LIN {X 0,Y 445.914,Z 450.872,A -85,B 0,C 180,E1 -16893.892,E2 -16893.892} C_VEL
LIN {X 0,Y 439.308,Z 442.238,A -85,B 0,C 180,E1 -16896.064,E2 -16896.064} C_VEL
LIN {X 0,Y 435.286,Z 437.114,A -85,B 0,C 180,E1 -16897.513,E2 -16897.513} C_VEL
LIN {X 0,Y 431.118,Z 431.872,A -85,B 0,C 180,E1 -16899.144,E2 -16899.144} C_VEL
LIN {X 0,Y 426.688,Z 426.377,A -85,B 0,C 180,E1 -16901.061,E2 -16901.061} C_VEL
LIN {X 0,Y 423.049,Z 422.011,A -85,B 0,C 180,E1 -16902.816,E2 -16902.816} C_VEL
LIN {X 0,Y 422.048,Z 420.717,A -85,B 0,C 180,E1 -16903.341,E2 -16903.341} C_VEL
LIN {X 0,Y 418.805,Z 417.442,A -85,B 0,C 180,E1 -16905.128,E2 -16905.128} C_VEL
LIN {X 0,Y 417.28,Z 414.785,A -85,B 0,C 180,E1 -16906.136,E2 -16906.136} C_VEL
LIN {X 0,Y 413.911,Z 412.07,A -85,B 0,C 180,E1 -16908.434,E2 -16908.434} C_VEL
LIN {X 0,Y 411.982,Z 408.411,A -85,B 0,C 180,E1 -16910.218,E2 -16910.218} C_VEL
LIN {X 0,Y 408.184,Z 405.747,A -85,B 0,C 180,E1 -16914.659,E2 -16914.659} C_VEL
LIN {X 0,Y 406.884,Z 403.015,A -85,B 0,C 180,E1 -16919.155,E2 -16919.155} C_VEL
LIN {X 0,Y 406.916,Z 403.188,A -85,B 0,C 180,E1 -16920.986,E2 -16920.986} C_VEL
LIN {X 0,Y 411.873,Z 408.41,A -85,B 0,C 180,E1 -16929.361,E2 -16929.361} C_VEL
LIN {X 0,Y 414.509,Z 412.704,A -85,B 0,C 180,E1 -16931.691,E2 -16931.691} C_VEL
LIN {X 0,Y 417.544,Z 415.253,A -85,B 0,C 180,E1 -16933.714,E2 -16933.714} C_VEL
LIN {X 0,Y 420.375,Z 419.282,A -85,B 0,C 180,E1 -16935.45,E2 -16935.45} C_VEL
LIN {X 0,Y 422.697,Z 421.438,A -85,B 0,C 180,E1 -16936.664,E2 -16936.664} C_VEL
LIN {X 0,Y 425.915,Z 425.709,A -85,B 0,C 180,E1 -16938.265,E2 -16938.265} C_VEL
LIN {X 0,Y 427.713,Z 427.589,A -85,B 0,C 180,E1 -16939.069,E2 -16939.069} C_VEL
LIN {X 0,Y 431.546,Z 432.247,A -85,B 0,C 180,E1 -16940.692,E2 -16940.692} C_VEL
LIN {X 0,Y 438.177,Z 440.986,A -85,B 0,C 180,E1 -16943.216,E2 -16943.216} C_VEL
LIN {X 0,Y 447.328,Z 454.311,A -85,B 0,C 180,E1 -16946.269,E2 -16946.269} C_VEL
LIN {X 0,Y 457.218,Z 469.808,A -85,B 0,C 180,E1 -16949.152,E2 -16949.152} C_VEL
LIN {X 0,Y 466.824,Z 485.963,A -85,B 0,C 180,E1 -16951.653,E2 -16951.653} C_VEL
LIN {X 0,Y 475.146,Z 500.955,A -85,B 0,C 180,E1 -16953.636,E2 -16953.636} C_VEL
LIN {X 0,Y 460.946,Z 747.179,A -85,B 0,C 180,E1 -16957.557,E2 -16957.557} C_VEL
LIN {X 0,Y 458.843,Z 772.183,A -85,B 0,C 180,E1 -16958.029,E2 -16958.029} C_VEL
LIN {X 0,Y 455.888,Z 795.416,A -85,B 0,C 180,E1 -16958.602,E2 -16958.602} C_VEL
LIN {X 0,Y 451.88,Z 819.021,A -85,B 0,C 180,E1 -16959.383,E2 -16959.383} C_VEL
LIN {X 0,Y 448.092,Z 837.848,A -85,B 0,C 180,E1 -16960.157,E2 -16960.157} C_VEL
LIN {X 0,Y 442.735,Z 861.158,A -85,B 0,C 180,E1 -16961.329,E2 -16961.329} C_VEL
LIN {X 0,Y 437.251,Z 881.76,A -85,B 0,C 180,E1 -16962.601,E2 -16962.601} C_VEL
LIN {X 0,Y 431.383,Z 901.908,A -85,B 0,C 180,E1 -16964.066,E2 -16964.066} C_VEL
LIN {X 0,Y 424.657,Z 922.896,A -85,B 0,C 180,E1 -16965.902,E2 -16965.902} C_VEL
LIN {X 0,Y 418.742,Z 940.201,A -85,B 0,C 180,E1 -16967.672,E2 -16967.672} C_VEL
LIN {X 0,Y 411.479,Z 960.285,A -85,B 0,C 180,E1 -16970.095,E2 -16970.095} C_VEL
LIN {X 0,Y 405.621,Z 975.927,A -85,B 0,C 180,E1 -16972.313,E2 -16972.313} C_VEL
LIN {X 0,Y 398.802,Z 993.871,A -85,B 0,C 180,E1 -16975.309,E2 -16975.309} C_VEL
LIN {X 0,Y 393.732,Z 1007.261,A -85,B 0,C 180,E1 -16977.943,E2 -16977.943} C_VEL
LIN {X 0,Y 388.289,Z 1022.091,A -85,B 0,C 180,E1 -16981.382,E2 -16981.382} C_VEL
LIN {X 0,Y 384.646,Z 1032.615,A -85,B 0,C 180,E1 -16984.271,E2 -16984.271} C_VEL
LIN {X 0,Y 381.229,Z 1043.573,A -85,B 0,C 180,E1 -16987.81,E2 -16987.81} C_VEL
LIN {X 0,Y 378.881,Z 1052.198,A -85,B 0,C 180,E1 -16991.218,E2 -16991.218} C_VEL
LIN {X 0,Y 377.283,Z 1059.672,A -85,B 0,C 180,E1 -16994.789,E2 -16994.789} C_VEL
LIN {X 0,Y 376.39,Z 1065.338,A -85,B 0,C 180,E1 -16998.352,E2 -16998.352} C_VEL
LIN {X 0,Y 376.05,Z 1069.072,A -85,B 0,C 180,E1 -17001.437,E2 -17001.437} C_VEL
LIN {X 0,Y 375.953,Z 1072.023,A -85,B 0,C 180,E1 -17004.965,E2 -17004.965} C_VEL
LIN {X 0,Y 375.957,Z 1073.297,A -85,B 0,C 180,E1 -17008.323,E2 -17008.323} C_VEL
LIN {X 0,Y 375.964,Z 1073.365,A -85,B 0,C 180,E1 -17011.219,E2 -17011.219} C_VEL
LIN {X 0,Y 375.948,Z 1072.423,A -85,B 0,C 180,E1 -17014.152,E2 -17014.152} C_VEL
LIN {X 0,Y 375.991,Z 1070.035,A -85,B 0,C 180,E1 -17017.641,E2 -17017.641} C_VEL
LIN {X 0,Y 376.318,Z 1065.955,A -85,B 0,C 180,E1 -17021.184,E2 -17021.184} C_VEL
LIN {X 0,Y 377.033,Z 1060.963,A -85,B 0,C 180,E1 -17024.435,E2 -17024.435} C_VEL
LIN {X 0,Y 378.625,Z 1053.245,A -85,B 0,C 180,E1 -17028.316,E2 -17028.316} C_VEL
LIN {X 0,Y 380.724,Z 1045.185,A -85,B 0,C 180,E1 -17031.572,E2 -17031.572} C_VEL
LIN {X 0,Y 383.966,Z 1034.661,A -85,B 0,C 180,E1 -17035.117,E2 -17035.117} C_VEL
LIN {X 0,Y 387.657,Z 1023.784,A -85,B 0,C 180,E1 -17038.165,E2 -17038.165} C_VEL
LIN {X 0,Y 392.448,Z 1010.715,A -85,B 0,C 180,E1 -17041.316,E2 -17041.316} C_VEL
LIN {X 0,Y 397.898,Z 996.124,A -85,B 0,C 180,E1 -17044.256,E2 -17044.256} C_VEL
LIN {X 0,Y 403.578,Z 981.252,A -85,B 0,C 180,E1 -17046.845,E2 -17046.845} C_VEL
LIN {X 0,Y 410.123,Z 963.744,A -85,B 0,C 180,E1 -17049.428,E2 -17049.428} C_VEL
LIN {X 0,Y 416.214,Z 947.095,A -85,B 0,C 180,E1 -17051.532,E2 -17051.532} C_VEL
LIN {X 0,Y 423.277,Z 926.792,A -85,B 0,C 180,E1 -17053.709,E2 -17053.709} C_VEL
LIN {X 0,Y 429.253,Z 908.409,A -85,B 0,C 180,E1 -17055.382,E2 -17055.382} C_VEL
LIN {X 0,Y 436.027,Z 885.844,A -85,B 0,C 180,E1 -17057.111,E2 -17057.111} C_VEL
LIN {X 0,Y 441.133,Z 866.944,A -85,B 0,C 180,E1 -17058.319,E2 -17058.319} C_VEL
LIN {X 0,Y 446.428,Z 845.202,A -85,B 0,C 180,E1 -17059.494,E2 -17059.494} C_VEL
LIN {X 0,Y 451.109,Z 822.479,A -85,B 0,C 180,E1 -17060.475,E2 -17060.475} C_VEL
LIN {X 0,Y 454.909,Z 800.788,A -85,B 0,C 180,E1 -17061.227,E2 -17061.227} C_VEL
LIN {X 0,Y 458.427,Z 774.973,A -85,B 0,C 180,E1 -17061.899,E2 -17061.899} C_VEL
LIN {X 0,Y 460.452,Z 752.549,A -85,B 0,C 180,E1 -17062.338,E2 -17062.338} C_VEL
LIN {X 0,Y 474.798,Z 504.728,A -85,B 0,C 180,E1 -17066.292,E2 -17066.292} C_VEL
LIN {X 0,Y 474.918,Z 500.686,A -85,B 0,C 180,E1 -17066.377,E2 -17066.377} C_VEL
LIN {X 0,Y 465.136,Z 483.112,A -85,B 0,C 180,E1 -17068.725,E2 -17068.725} C_VEL
LIN {X 0,Y 455.822,Z 467.629,A -85,B 0,C 180,E1 -17071.181,E2 -17071.181} C_VEL
LIN {X 0,Y 446.583,Z 453.314,A -85,B 0,C 180,E1 -17073.899,E2 -17073.899} C_VEL
LIN {X 0,Y 439.183,Z 442.658,A -85,B 0,C 180,E1 -17076.342,E2 -17076.342} C_VEL
LIN {X 0,Y 435.375,Z 437.187,A -85,B 0,C 180,E1 -17077.732,E2 -17077.732} C_VEL
LIN {X 0,Y 431.177,Z 431.925,A -85,B 0,C 180,E1 -17079.361,E2 -17079.361} C_VEL
LIN {X 0,Y 427.435,Z 427.213,A -85,B 0,C 180,E1 -17080.954,E2 -17080.954} C_VEL
LIN {X 0,Y 423.28,Z 422.498,A -85,B 0,C 180,E1 -17082.896,E2 -17082.896} C_VEL
LIN {X 0,Y 422.163,Z 420.799,A -85,B 0,C 180,E1 -17083.488,E2 -17083.488} C_VEL
LIN {X 0,Y 418.647,Z 417.219,A -85,B 0,C 180,E1 -17085.406,E2 -17085.406} C_VEL
LIN {X 0,Y 417.091,Z 414.724,A -85,B 0,C 180,E1 -17086.412,E2 -17086.412} C_VEL
LIN {X 0,Y 413.807,Z 411.904,A -85,B 0,C 180,E1 -17088.642,E2 -17088.642} C_VEL
LIN {X 0,Y 411.904,Z 408.425,A -85,B 0,C 180,E1 -17090.358,E2 -17090.358} C_VEL
LIN {X 0,Y 407.764,Z 405.265,A -85,B 0,C 180,E1 -17095.218,E2 -17095.218} C_VEL
LIN {X 0,Y 406.659,Z 401.868,A -85,B 0,C 180,E1 -17099.577,E2 -17099.577} C_VEL
LIN {X 0,Y 406.701,Z 402.227,A -85,B 0,C 180,E1 -17101.55,E2 -17101.55} C_VEL
LIN {X 0,Y 410.534,Z 407.839,A -85,B 0,C 180,E1 -17108.826,E2 -17108.826} C_VEL
LIN {X 0,Y 412.126,Z 408.762,A -85,B 0,C 180,E1 -17110.272,E2 -17110.272} C_VEL
LIN {X 0,Y 414.158,Z 412.402,A -85,B 0,C 180,E1 -17112.054,E2 -17112.054} C_VEL
LIN {X 0,Y 417.516,Z 415.258,A -85,B 0,C 180,E1 -17114.281,E2 -17114.281} C_VEL
LIN {X 0,Y 420.259,Z 419.245,A -85,B 0,C 180,E1 -17115.95,E2 -17115.95} C_VEL
LIN {X 0,Y 422.739,Z 421.532,A -85,B 0,C 180,E1 -17117.233,E2 -17117.233} C_VEL
LIN {X 0,Y 426.281,Z 426.044,A -85,B 0,C 180,E1 -17118.958,E2 -17118.958} C_VEL
LIN {X 0,Y 427.727,Z 427.665,A -85,B 0,C 180,E1 -17119.6,E2 -17119.6} C_VEL
LIN {X 0,Y 431.51,Z 432.267,A -85,B 0,C 180,E1 -17121.191,E2 -17121.191} C_VEL
LIN {X 0,Y 437.246,Z 439.664,A -85,B 0,C 180,E1 -17123.376,E2 -17123.376} C_VEL
LIN {X 0,Y 441.857,Z 445.634,A -85,B 0,C 180,E1 -17124.963,E2 -17124.963} C_VEL
LIN {X 0,Y 448.316,Z 454.069,A -85,B 0,C 180,E1 -17126.992,E2 -17126.992} C_VEL
LIN {X 0,Y 458.368,Z 468.203,A -85,B 0,C 180,E1 -17129.826,E2 -17129.826} C_VEL
LIN {X 0,Y 467.534,Z 481.985,A -85,B 0,C 180,E1 -17132.14,E2 -17132.14} C_VEL
LIN {X 0,Y 475.238,Z 494.264,A -85,B 0,C 180,E1 -17133.93,E2 -17133.93} C_VEL
LIN {X 0,Y 460.96,Z 738.871,A -85,B 0,C 180,E1 -17137.83,E2 -17137.83} C_VEL
LIN {X 0,Y 458.981,Z 760.833,A -85,B 0,C 180,E1 -17138.272,E2 -17138.272} C_VEL
LIN {X 0,Y 455.614,Z 786.437,A -85,B 0,C 180,E1 -17138.98,E2 -17138.98} C_VEL
LIN {X 0,Y 452.234,Z 806.44,A -85,B 0,C 180,E1 -17139.698,E2 -17139.698} C_VEL
LIN {X 0,Y 447.751,Z 829.084,A -85,B 0,C 180,E1 -17140.699,E2 -17140.699} C_VEL
LIN {X 0,Y 442.594,Z 850.765,A -85,B 0,C 180,E1 -17141.893,E2 -17141.893} C_VEL
LIN {X 0,Y 437.114,Z 871.313,A -85,B 0,C 180,E1 -17143.234,E2 -17143.234} C_VEL
LIN {X 0,Y 430.715,Z 892.744,A -85,B 0,C 180,E1 -17144.924,E2 -17144.924} C_VEL
LIN {X 0,Y 424.856,Z 910.758,A -85,B 0,C 180,E1 -17146.59,E2 -17146.59} C_VEL
LIN {X 0,Y 417.698,Z 931.227,A -85,B 0,C 180,E1 -17148.83,E2 -17148.83} C_VEL
LIN {X 0,Y 411.851,Z 947.019,A -85,B 0,C 180,E1 -17150.86,E2 -17150.86} C_VEL
LIN {X 0,Y 405.104,Z 964.603,A -85,B 0,C 180,E1 -17153.499,E2 -17153.499} C_VEL
LIN {X 0,Y 399.413,Z 979.074,A -85,B 0,C 180,E1 -17156.065,E2 -17156.065} C_VEL
LIN {X 0,Y 393.645,Z 993.854,A -85,B 0,C 180,E1 -17159.13,E2 -17159.13} C_VEL
LIN {X 0,Y 388.99,Z 1005.906,A -85,B 0,C 180,E1 -17162.107,E2 -17162.107} C_VEL
LIN {X 0,Y 384.833,Z 1017.408,A -85,B 0,C 180,E1 -17165.436,E2 -17165.436} C_VEL
LIN {X 0,Y 381.521,Z 1027.213,A -85,B 0,C 180,E1 -17168.909,E2 -17168.909} C_VEL
LIN {X 0,Y 379.086,Z 1035.65,A -85,B 0,C 180,E1 -17172.501,E2 -17172.501} C_VEL
LIN {X 0,Y 377.492,Z 1042.13,A -85,B 0,C 180,E1 -17176.052,E2 -17176.052} C_VEL
LIN {X 0,Y 376.627,Z 1046.785,A -85,B 0,C 180,E1 -17179.29,E2 -17179.29} C_VEL
LIN {X 0,Y 376.148,Z 1050.669,A -85,B 0,C 180,E1 -17183.13,E2 -17183.13} C_VEL
LIN {X 0,Y 376.009,Z 1052.533,A -85,B 0,C 180,E1 -17186.188,E2 -17186.188} C_VEL
LIN {X 0,Y 375.969,Z 1053.36,A -85,B 0,C 180,E1 -17189.238,E2 -17189.238} C_VEL
LIN {X 0,Y 375.985,Z 1053.045,A -85,B 0,C 180,E1 -17192.744,E2 -17192.744} C_VEL
LIN {X 0,Y 376.092,Z 1051.299,A -85,B 0,C 180,E1 -17196.105,E2 -17196.105} C_VEL
LIN {X 0,Y 376.366,Z 1048.637,A -85,B 0,C 180,E1 -17199.172,E2 -17199.172} C_VEL
LIN {X 0,Y 377.086,Z 1044.286,A -85,B 0,C 180,E1 -17202.714,E2 -17202.714} C_VEL
LIN {X 0,Y 378.398,Z 1038.227,A -85,B 0,C 180,E1 -17206.266,E2 -17206.266} C_VEL
LIN {X 0,Y 380.273,Z 1031.39,A -85,B 0,C 180,E1 -17209.508,E2 -17209.508} C_VEL
LIN {X 0,Y 383.325,Z 1021.762,A -85,B 0,C 180,E1 -17213.196,E2 -17213.196} C_VEL
LIN {X 0,Y 386.688,Z 1012.189,A -85,B 0,C 180,E1 -17216.242,E2 -17216.242} C_VEL
LIN {X 0,Y 388.467,Z 1007.407,A -85,B 0,C 180,E1 -17217.598,E2 -17217.598} C_VEL
LIN {X 0,Y 388.905,Z 1003.88,A -85,B 0,C 180,E1 -17218.615,E2 -17218.615} C_VEL
LIN {X 0,Y 387.122,Z 994.607,A -85,B 0,C 180,E1 -17221.427,E2 -17221.427} C_VEL
LIN {X 0,Y 387.838,Z 991.149,A -85,B 0,C 180,E1 -17222.262,E2 -17222.262} C_VEL
LIN {X 0,Y 393.105,Z 978.251,A -85,B 0,C 180,E1 -17224.911,E2 -17224.911} C_VEL
LIN {X 0,Y 399.46,Z 962.832,A -85,B 0,C 180,E1 -17227.644,E2 -17227.644} C_VEL
LIN {X 0,Y 406.146,Z 945.85,A -85,B 0,C 180,E1 -17230.167,E2 -17230.167} C_VEL
LIN {X 0,Y 412.721,Z 928.691,A -85,B 0,C 180,E1 -17232.36,E2 -17232.36} C_VEL
LIN {X 0,Y 419.697,Z 909.139,A -85,B 0,C 180,E1 -17234.462,E2 -17234.462} C_VEL
LIN {X 0,Y 425.918,Z 890.53,A -85,B 0,C 180,E1 -17236.168,E2 -17236.168} C_VEL
LIN {X 0,Y 432.407,Z 869.027,A -85,B 0,C 180,E1 -17237.827,E2 -17237.827} C_VEL
LIN {X 0,Y 437.827,Z 849.172,A -85,B 0,C 180,E1 -17239.106,E2 -17239.106} C_VEL
LIN {X 0,Y 443.66,Z 824.456,A -85,B 0,C 180,E1 -17240.424,E2 -17240.424} C_VEL
LIN {X 0,Y 447.87,Z 803.378,A -85,B 0,C 180,E1 -17241.327,E2 -17241.327} C_VEL
LIN {X 0,Y 452.017,Z 777.908,A -85,B 0,C 180,E1 -17242.186,E2 -17242.186} C_VEL
LIN {X 0,Y 454.733,Z 755.827,A -85,B 0,C 180,E1 -17242.742,E2 -17242.742} C_VEL
LIN {X 0,Y 456.958,Z 728.166,A -85,B 0,C 180,E1 -17243.252,E2 -17243.252} C_VEL
LIN {X 0,Y 470.68,Z 498.278,A -85,B 0,C 180,E1 -17246.928,E2 -17246.928} C_VEL
LIN {X 0,Y 460.809,Z 482.688,A -85,B 0,C 180,E1 -17249.342,E2 -17249.342} C_VEL
LIN {X 0,Y 451.523,Z 469.038,A -85,B 0,C 180,E1 -17251.856,E2 -17251.856} C_VEL
LIN {X 0,Y 443.324,Z 457.626,A -85,B 0,C 180,E1 -17254.339,E2 -17254.339} C_VEL
LIN {X 0,Y 436.928,Z 449.186,A -85,B 0,C 180,E1 -17256.499,E2 -17256.499} C_VEL
LIN {X 0,Y 433.152,Z 444.297,A -85,B 0,C 180,E1 -17257.897,E2 -17257.897} C_VEL
LIN {X 0,Y 429.218,Z 439.263,A -85,B 0,C 180,E1 -17259.476,E2 -17259.476} C_VEL
LIN {X 0,Y 425.01,Z 433.941,A -85,B 0,C 180,E1 -17261.34,E2 -17261.34} C_VEL
LIN {X 0,Y 421.316,Z 429.373,A -85,B 0,C 180,E1 -17263.17,E2 -17263.17} C_VEL
LIN {X 0,Y 420.319,Z 428.242,A -85,B 0,C 180,E1 -17263.697,E2 -17263.697} C_VEL
LIN {X 0,Y 417.071,Z 424.661,A -85,B 0,C 180,E1 -17265.562,E2 -17265.562} C_VEL
LIN {X 0,Y 415.885,Z 422.55,A -85,B 0,C 180,E1 -17266.372,E2 -17266.372} C_VEL
LIN {X 0,Y 412.595,Z 419.762,A -85,B 0,C 180,E1 -17268.679,E2 -17268.679} C_VEL
LIN {X 0,Y 410.702,Z 416.259,A -85,B 0,C 180,E1 -17270.471,E2 -17270.471} C_VEL
LIN {X 0,Y 406.544,Z 412.767,A -85,B 0,C 180,E1 -17276.051,E2 -17276.051} C_VEL
LIN {X 0,Y 405.909,Z 410.957,A -85,B 0,C 180,E1 -17279.153,E2 -17279.153} C_VEL
LIN {X 0,Y 405.928,Z 411.083,A -85,B 0,C 180,E1 -17280.847,E2 -17280.847} C_VEL
LIN {X 0,Y 410.888,Z 416.54,A -85,B 0,C 180,E1 -17289.384,E2 -17289.384} C_VEL
LIN {X 0,Y 413,Z 420.204,A -85,B 0,C 180,E1 -17291.309,E2 -17291.309} C_VEL
LIN {X 0,Y 416.144,Z 423,A -85,B 0,C 180,E1 -17293.478,E2 -17293.478} C_VEL
LIN {X 0,Y 419.168,Z 427.21,A -85,B 0,C 180,E1 -17295.354,E2 -17295.354} C_VEL
LIN {X 0,Y 421.152,Z 429.131,A -85,B 0,C 180,E1 -17296.411,E2 -17296.411} C_VEL
LIN {X 0,Y 424.53,Z 433.532,A -85,B 0,C 180,E1 -17298.113,E2 -17298.113} C_VEL
LIN {X 0,Y 426.083,Z 435.288,A -85,B 0,C 180,E1 -17298.825,E2 -17298.825} C_VEL
LIN {X 0,Y 430.863,Z 441.312,A -85,B 0,C 180,E1 -17300.869,E2 -17300.869} C_VEL
LIN {X 0,Y 436.072,Z 448.276,A -85,B 0,C 180,E1 -17302.871,E2 -17302.871} C_VEL
LIN {X 0,Y 444.894,Z 461.347,A -85,B 0,C 180,E1 -17305.886,E2 -17305.886} C_VEL
LIN {X 0,Y 454.529,Z 476.71,A -85,B 0,C 180,E1 -17308.765,E2 -17308.765} C_VEL
LIN {X 0,Y 463.774,Z 492.562,A -85,B 0,C 180,E1 -17311.233,E2 -17311.233} C_VEL
LIN {X 0,Y 470.494,Z 504.94,A -85,B 0,C 180,E1 -17312.89,E2 -17312.89} C_VEL
LIN {X 0,Y 455.687,Z 752.602,A -85,B 0,C 180,E1 -17316.856,E2 -17316.856} C_VEL
LIN {X 0,Y 453.608,Z 774.959,A -85,B 0,C 180,E1 -17317.295,E2 -17317.295} C_VEL
LIN {X 0,Y 449.936,Z 801.11,A -85,B 0,C 180,E1 -17317.979,E2 -17317.979} C_VEL
LIN {X 0,Y 446.231,Z 821.754,A -85,B 0,C 180,E1 -17318.695,E2 -17318.695} C_VEL
LIN {X 0,Y 441.541,Z 844.082,A -85,B 0,C 180,E1 -17319.651,E2 -17319.651} C_VEL
LIN {X 0,Y 436.07,Z 865.993,A -85,B 0,C 180,E1 -17320.828,E2 -17320.828} C_VEL
LIN {X 0,Y 430.554,Z 885.873,A -85,B 0,C 180,E1 -17322.099,E2 -17322.099} C_VEL
LIN {X 0,Y 423.78,Z 907.768,A -85,B 0,C 180,E1 -17323.781,E2 -17323.781} C_VEL
LIN {X 0,Y 417.835,Z 925.512,A -85,B 0,C 180,E1 -17325.396,E2 -17325.396} C_VEL
LIN {X 0,Y 410.636,Z 945.656,A -85,B 0,C 180,E1 -17327.545,E2 -17327.545} C_VEL
LIN {X 0,Y 404.194,Z 962.624,A -85,B 0,C 180,E1 -17329.692,E2 -17329.692} C_VEL
LIN {X 0,Y 397.689,Z 979.441,A -85,B 0,C 180,E1 -17332.159,E2 -17332.159} C_VEL
LIN {X 0,Y 391.391,Z 995.21,A -85,B 0,C 180,E1 -17334.914,E2 -17334.914} C_VEL
LIN {X 0,Y 385.92,Z 1009.168,A -85,B 0,C 180,E1 -17337.742,E2 -17337.742} C_VEL
LIN {X 0,Y 380.726,Z 1022.659,A -85,B 0,C 180,E1 -17340.992,E2 -17340.992} C_VEL
LIN {X 0,Y 376.742,Z 1033.729,A -85,B 0,C 180,E1 -17344.122,E2 -17344.122} C_VEL
LIN {X 0,Y 373.191,Z 1044.59,A -85,B 0,C 180,E1 -17347.804,E2 -17347.804} C_VEL
LIN {X 0,Y 370.916,Z 1052.699,A -85,B 0,C 180,E1 -17351.126,E2 -17351.126} C_VEL
LIN {X 0,Y 369.175,Z 1060.507,A -85,B 0,C 180,E1 -17355.09,E2 -17355.09} C_VEL
LIN {X 0,Y 368.378,Z 1065.544,A -85,B 0,C 180,E1 -17358.413,E2 -17358.413} C_VEL
LIN {X 0,Y 368.014,Z 1069.51,A -85,B 0,C 180,E1 -17361.878,E2 -17361.878} C_VEL
LIN {X 0,Y 367.95,Z 1072.091,A -85,B 0,C 180,E1 -17365.48,E2 -17365.48} C_VEL
LIN {X 0,Y 367.963,Z 1073.13,A -85,B 0,C 180,E1 -17368.598,E2 -17368.598} C_VEL
LIN {X 0,Y 367.963,Z 1073.128,A -85,B 0,C 180,E1 -17371.401,E2 -17371.401} C_VEL
LIN {X 0,Y 367.951,Z 1072.084,A -85,B 0,C 180,E1 -17374.52,E2 -17374.52} C_VEL
LIN {X 0,Y 368.026,Z 1069.332,A -85,B 0,C 180,E1 -17378.279,E2 -17378.279} C_VEL
LIN {X 0,Y 368.378,Z 1065.527,A -85,B 0,C 180,E1 -17381.587,E2 -17381.587} C_VEL
LIN {X 0,Y 369.173,Z 1060.484,A -85,B 0,C 180,E1 -17384.91,E2 -17384.91} C_VEL
LIN {X 0,Y 370.917,Z 1052.653,A -85,B 0,C 180,E1 -17388.879,E2 -17388.879} C_VEL
LIN {X 0,Y 373.188,Z 1044.552,A -85,B 0,C 180,E1 -17392.196,E2 -17392.196} C_VEL
LIN {X 0,Y 376.835,Z 1033.394,A -85,B 0,C 180,E1 -17395.964,E2 -17395.964} C_VEL
LIN {X 0,Y 380.796,Z 1022.397,A -85,B 0,C 180,E1 -17399.063,E2 -17399.063} C_VEL
LIN {X 0,Y 386.228,Z 1008.248,A -85,B 0,C 180,E1 -17402.438,E2 -17402.438} C_VEL
LIN {X 0,Y 391.38,Z 995.121,A -85,B 0,C 180,E1 -17405.087,E2 -17405.087} C_VEL
LIN {X 0,Y 397.755,Z 979.124,A -85,B 0,C 180,E1 -17407.875,E2 -17407.875} C_VEL
LIN {X 0,Y 404.373,Z 961.987,A -85,B 0,C 180,E1 -17410.379,E2 -17410.379} C_VEL
LIN {X 0,Y 411.394,Z 943.499,A -85,B 0,C 180,E1 -17412.696,E2 -17412.696} C_VEL
LIN {X 0,Y 418.071,Z 924.575,A -85,B 0,C 180,E1 -17414.68,E2 -17414.68} C_VEL
LIN {X 0,Y 424.248,Z 906.082,A -85,B 0,C 180,E1 -17416.349,E2 -17416.349} C_VEL
LIN {X 0,Y 431.041,Z 883.812,A -85,B 0,C 180,E1 -17418.027,E2 -17418.027} C_VEL
LIN {X 0,Y 436.285,Z 864.804,A -85,B 0,C 180,E1 -17419.23,E2 -17419.23} C_VEL
LIN {X 0,Y 442.064,Z 841.142,A -85,B 0,C 180,E1 -17420.47,E2 -17420.47} C_VEL
LIN {X 0,Y 446.283,Z 820.92,A -85,B 0,C 180,E1 -17421.324,E2 -17421.324} C_VEL
LIN {X 0,Y 450.329,Z 798.213,A -85,B 0,C 180,E1 -17422.098,E2 -17422.098} C_VEL
LIN {X 0,Y 453.635,Z 773.646,A -85,B 0,C 180,E1 -17422.722,E2 -17422.722} C_VEL
LIN {X 0,Y 455.717,Z 750.597,A -85,B 0,C 180,E1 -17423.168,E2 -17423.168} C_VEL
LIN {X 0,Y 470.369,Z 504.718,A -85,B 0,C 180,E1 -17427.103,E2 -17427.103} C_VEL
LIN {X 0,Y 461.156,Z 488.101,A -85,B 0,C 180,E1 -17429.393,E2 -17429.393} C_VEL
LIN {X 0,Y 452.739,Z 473.897,A -85,B 0,C 180,E1 -17431.687,E2 -17431.687} C_VEL
LIN {X 0,Y 443.971,Z 460.049,A -85,B 0,C 180,E1 -17434.343,E2 -17434.343} C_VEL
LIN {X 0,Y 435.136,Z 446.928,A -85,B 0,C 180,E1 -17437.398,E2 -17437.398} C_VEL
LIN {X 0,Y 429.267,Z 439.317,A -85,B 0,C 180,E1 -17439.692,E2 -17439.692} C_VEL
LIN {X 0,Y 424.878,Z 433.867,A -85,B 0,C 180,E1 -17441.618,E2 -17441.618} C_VEL
LIN {X 0,Y 421.348,Z 429.558,A -85,B 0,C 180,E1 -17443.348,E2 -17443.348} C_VEL
LIN {X 0,Y 420.422,Z 428.32,A -85,B 0,C 180,E1 -17443.843,E2 -17443.843} C_VEL
LIN {X 0,Y 416.907,Z 424.438,A -85,B 0,C 180,E1 -17445.84,E2 -17445.84} C_VEL
LIN {X 0,Y 415.691,Z 422.489,A -85,B 0,C 180,E1 -17446.649,E2 -17446.649} C_VEL
LIN {X 0,Y 412.399,Z 419.482,A -85,B 0,C 180,E1 -17448.957,E2 -17448.957} C_VEL
LIN {X 0,Y 410.616,Z 416.27,A -85,B 0,C 180,E1 -17450.61,E2 -17450.61} C_VEL
LIN {X 0,Y 406.578,Z 412.906,A -85,B 0,C 180,E1 -17455.628,E2 -17455.628} C_VEL
LIN {X 0,Y 405.68,Z 409.842,A -85,B 0,C 180,E1 -17459.576,E2 -17459.576} C_VEL
LIN {X 0,Y 405.712,Z 410.106,A -85,B 0,C 180,E1 -17461.412,E2 -17461.412} C_VEL
LIN {X 0,Y 409.428,Z 415.727,A -85,B 0,C 180,E1 -17468.709,E2 -17468.709} C_VEL
LIN {X 0,Y 410.848,Z 416.485,A -85,B 0,C 180,E1 -17470.021,E2 -17470.021} C_VEL
LIN {X 0,Y 412.915,Z 420.204,A -85,B 0,C 180,E1 -17471.878,E2 -17471.878} C_VEL
LIN {X 0,Y 416.11,Z 423.018,A -85,B 0,C 180,E1 -17474.046,E2 -17474.046} C_VEL
LIN {X 0,Y 418.931,Z 427.055,A -85,B 0,C 180,E1 -17475.789,E2 -17475.789} C_VEL
LIN {X 0,Y 421.124,Z 429.106,A -85,B 0,C 180,E1 -17476.945,E2 -17476.945} C_VEL
LIN {X 0,Y 424.749,Z 433.733,A -85,B 0,C 180,E1 -17478.744,E2 -17478.744} C_VEL
LIN {X 0,Y 426.232,Z 435.587,A -85,B 0,C 180,E1 -17479.422,E2 -17479.422} C_VEL
LIN {X 0,Y 430.751,Z 441.257,A -85,B 0,C 180,E1 -17481.338,E2 -17481.338} C_VEL
LIN {X 0,Y 435.325,Z 447.163,A -85,B 0,C 180,E1 -17483.091,E2 -17483.091} C_VEL
LIN {X 0,Y 439.784,Z 453.022,A -85,B 0,C 180,E1 -17484.658,E2 -17484.658} C_VEL
LIN {X 0,Y 446.154,Z 461.528,A -85,B 0,C 180,E1 -17486.702,E2 -17486.702} C_VEL
LIN {X 0,Y 455.667,Z 475.098,A -85,B 0,C 180,E1 -17489.442,E2 -17489.442} C_VEL
LIN {X 0,Y 464.596,Z 488.732,A -85,B 0,C 180,E1 -17491.75,E2 -17491.75} C_VEL
LIN {X 0,Y 470.567,Z 498.521,A -85,B 0,C 180,E1 -17493.185,E2 -17493.185} C_VEL
LIN {X 0,Y 456.03,Z 739.962,A -85,B 0,C 180,E1 -17497.051,E2 -17497.051} C_VEL
LIN {X 0,Y 453.931,Z 762.36,A -85,B 0,C 180,E1 -17497.509,E2 -17497.509} C_VEL
LIN {X 0,Y 450.491,Z 787.419,A -85,B 0,C 180,E1 -17498.213,E2 -17498.213} C_VEL
LIN {X 0,Y 446.939,Z 807.793,A -85,B 0,C 180,E1 -17498.951,E2 -17498.951} C_VEL
LIN {X 0,Y 442.004,Z 831.567,A -85,B 0,C 180,E1 -17500.027,E2 -17500.027} C_VEL
LIN {X 0,Y 436.988,Z 851.987,A -85,B 0,C 180,E1 -17501.167,E2 -17501.167} C_VEL
LIN {X 0,Y 431.168,Z 873.165,A -85,B 0,C 180,E1 -17502.566,E2 -17502.566} C_VEL
LIN {X 0,Y 424.786,Z 893.696,A -85,B 0,C 180,E1 -17504.213,E2 -17504.213} C_VEL
LIN {X 0,Y 418.538,Z 912.306,A -85,B 0,C 180,E1 -17505.957,E2 -17505.957} C_VEL
LIN {X 0,Y 411.588,Z 931.449,A -85,B 0,C 180,E1 -17508.082,E2 -17508.082} C_VEL
LIN {X 0,Y 405.54,Z 947.241,A -85,B 0,C 180,E1 -17510.13,E2 -17510.13} C_VEL
LIN {X 0,Y 398.547,Z 964.825,A -85,B 0,C 180,E1 -17512.798,E2 -17512.798} C_VEL
LIN {X 0,Y 392.824,Z 978.808,A -85,B 0,C 180,E1 -17515.302,E2 -17515.302} C_VEL
LIN {X 0,Y 387.149,Z 992.814,A -85,B 0,C 180,E1 -17518.206,E2 -17518.206} C_VEL
LIN {X 0,Y 381.968,Z 1005.562,A -85,B 0,C 180,E1 -17521.377,E2 -17521.377} C_VEL
LIN {X 0,Y 377.562,Z 1017.157,A -85,B 0,C 180,E1 -17524.763,E2 -17524.763} C_VEL
LIN {X 0,Y 373.976,Z 1027.157,A -85,B 0,C 180,E1 -17528.348,E2 -17528.348} C_VEL
LIN {X 0,Y 371.396,Z 1035.54,A -85,B 0,C 180,E1 -17531.965,E2 -17531.965} C_VEL
LIN {X 0,Y 369.667,Z 1042.099,A -85,B 0,C 180,E1 -17535.591,E2 -17535.591} C_VEL
LIN {X 0,Y 368.714,Z 1046.799,A -85,B 0,C 180,E1 -17538.899,E2 -17538.899} C_VEL
LIN {X 0,Y 368.179,Z 1050.773,A -85,B 0,C 180,E1 -17542.824,E2 -17542.824} C_VEL
LIN {X 0,Y 368.014,Z 1052.747,A -85,B 0,C 180,E1 -17546.105,E2 -17546.105} C_VEL
LIN {X 0,Y 367.972,Z 1053.574,A -85,B 0,C 180,E1 -17549.222,E2 -17549.222} C_VEL
LIN {X 0,Y 367.99,Z 1053.259,A -85,B 0,C 180,E1 -17552.804,E2 -17552.804} C_VEL
LIN {X 0,Y 368.107,Z 1051.513,A -85,B 0,C 180,E1 -17556.238,E2 -17556.238} C_VEL
LIN {X 0,Y 368.397,Z 1048.852,A -85,B 0,C 180,E1 -17559.372,E2 -17559.372} C_VEL
LIN {X 0,Y 369.177,Z 1044.501,A -85,B 0,C 180,E1 -17562.991,E2 -17562.991} C_VEL
LIN {X 0,Y 370.625,Z 1038.261,A -85,B 0,C 180,E1 -17566.716,E2 -17566.716} C_VEL
LIN {X 0,Y 372.797,Z 1030.914,A -85,B 0,C 180,E1 -17570.243,E2 -17570.243} C_VEL
LIN {X 0,Y 375.945,Z 1021.528,A -85,B 0,C 180,E1 -17573.846,E2 -17573.846} C_VEL
LIN {X 0,Y 379.536,Z 1011.9,A -85,B 0,C 180,E1 -17576.945,E2 -17576.945} C_VEL
LIN {X 0,Y 384.689,Z 998.86,A -85,B 0,C 180,E1 -17580.454,E2 -17580.454} C_VEL
LIN {X 0,Y 387.838,Z 991.149,A -85,B 0,C 180,E1 -17582.262,E2 -17582.262} C_VEL
LIN {X 0,Y 388.647,Z 987.062,A -85,B 0,C 180,E1 -17583.23,E2 -17583.23} C_VEL
LIN {X 0,Y 387.965,Z 976.484,A -85,B 0,C 180,E1 -17585.946,E2 -17585.946} C_VEL
LIN {X 0,Y 388.953,Z 972.574,A -85,B 0,C 180,E1 -17586.727,E2 -17586.727} C_VEL
LIN {X 0,Y 395.372,Z 957.167,A -85,B 0,C 180,E1 -17589.297,E2 -17589.297} C_VEL
LIN {X 0,Y 402.403,Z 940.031,A -85,B 0,C 180,E1 -17591.754,E2 -17591.754} C_VEL
LIN {X 0,Y 409.338,Z 921.923,A -85,B 0,C 180,E1 -17593.926,E2 -17593.926} C_VEL
LIN {X 0,Y 415.99,Z 903.645,A -85,B 0,C 180,E1 -17595.808,E2 -17595.808} C_VEL
LIN {X 0,Y 422.699,Z 883.412,A -85,B 0,C 180,E1 -17597.564,E2 -17597.564} C_VEL
LIN {X 0,Y 428.338,Z 864.757,A -85,B 0,C 180,E1 -17598.938,E2 -17598.938} C_VEL
LIN {X 0,Y 434.494,Z 842.11,A -85,B 0,C 180,E1 -17600.334,E2 -17600.334} C_VEL
LIN {X 0,Y 439.137,Z 822.103,A -85,B 0,C 180,E1 -17601.351,E2 -17601.351} C_VEL
LIN {X 0,Y 443.644,Z 799.755,A -85,B 0,C 180,E1 -17602.287,E2 -17602.287} C_VEL
LIN {X 0,Y 447.503,Z 775.515,A -85,B 0,C 180,E1 -17603.07,E2 -17603.07} C_VEL
LIN {X 0,Y 450.28,Z 752.875,A -85,B 0,C 180,E1 -17603.623,E2 -17603.623} C_VEL
LIN {X 0,Y 452.761,Z 719.205,A -85,B 0,C 180,E1 -17604.212,E2 -17604.212} C_VEL
LIN {X 0,Y 466.087,Z 502.45,A -85,B 0,C 180,E1 -17607.692,E2 -17607.692} C_VEL
LIN {X 0,Y 456.767,Z 487.669,A -85,B 0,C 180,E1 -17610.059,E2 -17610.059} C_VEL
LIN {X 0,Y 448.611,Z 475.507,A -85,B 0,C 180,E1 -17612.344,E2 -17612.344} C_VEL
LIN {X 0,Y 439.77,Z 462.888,A -85,B 0,C 180,E1 -17615.126,E2 -17615.126} C_VEL
LIN {X 0,Y 431.692,Z 452.209,A -85,B 0,C 180,E1 -17618.033,E2 -17618.033} C_VEL
LIN {X 0,Y 427.179,Z 446.49,A -85,B 0,C 180,E1 -17619.874,E2 -17619.874} C_VEL
LIN {X 0,Y 423.202,Z 441.367,A -85,B 0,C 180,E1 -17621.685,E2 -17621.685} C_VEL
LIN {X 0,Y 419.482,Z 436.53,A -85,B 0,C 180,E1 -17623.593,E2 -17623.593} C_VEL
LIN {X 0,Y 415.677,Z 432.388,A -85,B 0,C 180,E1 -17625.789,E2 -17625.789} C_VEL
LIN {X 0,Y 414.285,Z 430.177,A -85,B 0,C 180,E1 -17626.745,E2 -17626.745} C_VEL
LIN {X 0,Y 411.126,Z 427.22,A -85,B 0,C 180,E1 -17629.065,E2 -17629.065} C_VEL
LIN {X 0,Y 409.584,Z 424.159,A -85,B 0,C 180,E1 -17630.586,E2 -17630.586} C_VEL
LIN {X 0,Y 405.418,Z 420.428,A -85,B 0,C 180,E1 -17636.465,E2 -17636.465} C_VEL
LIN {X 0,Y 404.925,Z 418.879,A -85,B 0,C 180,E1 -17639.293,E2 -17639.293} C_VEL
LIN {X 0,Y 404.963,Z 419.096,A -85,B 0,C 180,E1 -17640.99,E2 -17640.99} C_VEL
LIN {X 0,Y 409.687,Z 424.419,A -85,B 0,C 180,E1 -17649.199,E2 -17649.199} C_VEL
LIN {X 0,Y 411.85,Z 428.103,A -85,B 0,C 180,E1 -17651.199,E2 -17651.199} C_VEL
LIN {X 0,Y 414.752,Z 430.738,A -85,B 0,C 180,E1 -17653.24,E2 -17653.24} C_VEL
LIN {X 0,Y 417.844,Z 435.017,A -85,B 0,C 180,E1 -17655.191,E2 -17655.191} C_VEL
LIN {X 0,Y 419.669,Z 436.906,A -85,B 0,C 180,E1 -17656.186,E2 -17656.186} C_VEL
LIN {X 0,Y 423.148,Z 441.352,A -85,B 0,C 180,E1 -17657.961,E2 -17657.961} C_VEL
LIN {X 0,Y 424.804,Z 443.496,A -85,B 0,C 180,E1 -17658.741,E2 -17658.741} C_VEL
LIN {X 0,Y 429.099,Z 448.903,A -85,B 0,C 180,E1 -17660.601,E2 -17660.601} C_VEL
LIN {X 0,Y 433.904,Z 455.426,A -85,B 0,C 180,E1 -17662.491,E2 -17662.491} C_VEL
LIN {X 0,Y 442.48,Z 468.381,A -85,B 0,C 180,E1 -17665.498,E2 -17665.498} C_VEL
LIN {X 0,Y 451.863,Z 483.608,A -85,B 0,C 180,E1 -17668.373,E2 -17668.373} C_VEL
LIN {X 0,Y 460.858,Z 499.358,A -85,B 0,C 180,E1 -17670.836,E2 -17670.836} C_VEL
LIN {X 0,Y 465.915,Z 508.893,A -85,B 0,C 180,E1 -17672.126,E2 -17672.126} C_VEL
LIN {X 0,Y 450.766,Z 754.339,A -85,B 0,C 180,E1 -17676.074,E2 -17676.074} C_VEL
LIN {X 0,Y 448.507,Z 777.221,A -85,B 0,C 180,E1 -17676.532,E2 -17676.532} C_VEL
LIN {X 0,Y 444.729,Z 802.601,A -85,B 0,C 180,E1 -17677.216,E2 -17677.216} C_VEL
LIN {X 0,Y 440.753,Z 823.966,A -85,B 0,C 180,E1 -17677.97,E2 -17677.97} C_VEL
LIN {X 0,Y 435.265,Z 848.435,A -85,B 0,C 180,E1 -17679.063,E2 -17679.063} C_VEL
LIN {X 0,Y 430.062,Z 868.528,A -85,B 0,C 180,E1 -17680.174,E2 -17680.174} C_VEL
LIN {X 0,Y 423.534,Z 890.939,A -85,B 0,C 180,E1 -17681.659,E2 -17681.659} C_VEL
LIN {X 0,Y 417.166,Z 910.511,A -85,B 0,C 180,E1 -17683.227,E2 -17683.227} C_VEL
LIN {X 0,Y 410.188,Z 930.575,A -85,B 0,C 180,E1 -17685.114,E2 -17685.114} C_VEL
LIN {X 0,Y 402.968,Z 949.596,A -85,B 0,C 180,E1 -17687.263,E2 -17687.263} C_VEL
LIN {X 0,Y 395.944,Z 967.518,A -85,B 0,C 180,E1 -17689.628,E2 -17689.628} C_VEL
LIN {X 0,Y 389.027,Z 984.357,A -85,B 0,C 180,E1 -17692.286,E2 -17692.286} C_VEL
LIN {X 0,Y 383.062,Z 998.886,A -85,B 0,C 180,E1 -17694.952,E2 -17694.952} C_VEL
LIN {X 0,Y 377.025,Z 1013.557,A -85,B 0,C 180,E1 -17698.146,E2 -17698.146} C_VEL
LIN {X 0,Y 372.452,Z 1025.139,A -85,B 0,C 180,E1 -17701.103,E2 -17701.103} C_VEL
LIN {X 0,Y 367.816,Z 1037.64,A -85,B 0,C 180,E1 -17704.908,E2 -17704.908} C_VEL
LIN {X 0,Y 364.896,Z 1046.432,A -85,B 0,C 180,E1 -17708.12,E2 -17708.12} C_VEL
LIN {X 0,Y 362.428,Z 1055.22,A -85,B 0,C 180,E1 -17712.001,E2 -17712.001} C_VEL
LIN {X 0,Y 361.069,Z 1061.329,A -85,B 0,C 180,E1 -17715.404,E2 -17715.404} C_VEL
LIN {X 0,Y 360.289,Z 1066.384,A -85,B 0,C 180,E1 -17718.96,E2 -17718.96} C_VEL
LIN {X 0,Y 359.992,Z 1070.213,A -85,B 0,C 180,E1 -17722.82,E2 -17722.82} C_VEL
LIN {X 0,Y 359.951,Z 1072.157,A -85,B 0,C 180,E1 -17726.018,E2 -17726.018} C_VEL
LIN {X 0,Y 359.972,Z 1072.987,A -85,B 0,C 180,E1 -17729.045,E2 -17729.045} C_VEL
LIN {X 0,Y 359.963,Z 1072.749,A -85,B 0,C 180,E1 -17732.547,E2 -17732.547} C_VEL
LIN {X 0,Y 359.965,Z 1070.902,A -85,B 0,C 180,E1 -17736.219,E2 -17736.219} C_VEL
LIN {X 0,Y 360.102,Z 1068.135,A -85,B 0,C 180,E1 -17739.429,E2 -17739.429} C_VEL
LIN {X 0,Y 360.677,Z 1063.617,A -85,B 0,C 180,E1 -17743.14,E2 -17743.14} C_VEL
LIN {X 0,Y 361.891,Z 1057.355,A -85,B 0,C 180,E1 -17746.864,E2 -17746.864} C_VEL
LIN {X 0,Y 363.732,Z 1050.284,A -85,B 0,C 180,E1 -17750.265,E2 -17750.265} C_VEL
LIN {X 0,Y 366.847,Z 1040.393,A -85,B 0,C 180,E1 -17754.132,E2 -17754.132} C_VEL
LIN {X 0,Y 370.419,Z 1030.407,A -85,B 0,C 180,E1 -17757.366,E2 -17757.366} C_VEL
LIN {X 0,Y 375.491,Z 1017.348,A -85,B 0,C 180,E1 -17760.926,E2 -17760.926} C_VEL
LIN {X 0,Y 380.624,Z 1004.614,A -85,B 0,C 180,E1 -17763.843,E2 -17763.843} C_VEL
LIN {X 0,Y 386.95,Z 989.376,A -85,B 0,C 180,E1 -17766.834,E2 -17766.834} C_VEL
LIN {X 0,Y 393.412,Z 973.505,A -85,B 0,C 180,E1 -17769.449,E2 -17769.449} C_VEL
LIN {X 0,Y 400.429,Z 956.104,A -85,B 0,C 180,E1 -17771.916,E2 -17771.916} C_VEL
LIN {X 0,Y 407.606,Z 937.15,A -85,B 0,C 180,E1 -17774.161,E2 -17774.161} C_VEL
LIN {X 0,Y 414.688,Z 917.629,A -85,B 0,C 180,E1 -17776.132,E2 -17776.132} C_VEL
LIN {X 0,Y 421.427,Z 897.163,A -85,B 0,C 180,E1 -17777.855,E2 -17777.855} C_VEL
LIN {X 0,Y 427.51,Z 877.258,A -85,B 0,C 180,E1 -17779.27,E2 -17779.27} C_VEL
LIN {X 0,Y 433.813,Z 853.771,A -85,B 0,C 180,E1 -17780.65,E2 -17780.65} C_VEL
LIN {X 0,Y 438.827,Z 832.475,A -85,B 0,C 180,E1 -17781.669,E2 -17781.669} C_VEL
LIN {X 0,Y 443.84,Z 807.02,A -85,B 0,C 180,E1 -17782.632,E2 -17782.632} C_VEL
LIN {X 0,Y 447.306,Z 785.214,A -85,B 0,C 180,E1 -17783.262,E2 -17783.262} C_VEL
LIN {X 0,Y 450.322,Z 758.412,A -85,B 0,C 180,E1 -17783.841,E2 -17783.841} C_VEL
LIN {X 0,Y 464.242,Z 532.943,A -85,B 0,C 180,E1 -17787.481,E2 -17787.481} C_VEL
LIN {X 0,Y 465.723,Z 508.479,A -85,B 0,C 180,E1 -17787.883,E2 -17787.883} C_VEL
LIN {X 0,Y 456.452,Z 491.601,A -85,B 0,C 180,E1 -17790.289,E2 -17790.289} C_VEL
LIN {X 0,Y 448.306,Z 477.905,A -85,B 0,C 180,E1 -17792.612,E2 -17792.612} C_VEL
LIN {X 0,Y 440.298,Z 465.056,A -85,B 0,C 180,E1 -17795.157,E2 -17795.157} C_VEL
LIN {X 0,Y 431.833,Z 452.512,A -85,B 0,C 180,E1 -17798.219,E2 -17798.219} C_VEL
LIN {X 0,Y 427.218,Z 446.549,A -85,B 0,C 180,E1 -17800.09,E2 -17800.09} C_VEL
LIN {X 0,Y 423.064,Z 441.297,A -85,B 0,C 180,E1 -17801.964,E2 -17801.964} C_VEL
LIN {X 0,Y 419.503,Z 436.713,A -85,B 0,C 180,E1 -17803.772,E2 -17803.772} C_VEL
LIN {X 0,Y 415.193,Z 431.641,A -85,B 0,C 180,E1 -17806.278,E2 -17806.278} C_VEL
LIN {X 0,Y 414.299,Z 430.246,A -85,B 0,C 180,E1 -17806.887,E2 -17806.887} C_VEL
LIN {X 0,Y 411.005,Z 427.057,A -85,B 0,C 180,E1 -17809.274,E2 -17809.274} C_VEL
LIN {X 0,Y 409.337,Z 424.104,A -85,B 0,C 180,E1 -17810.864,E2 -17810.864} C_VEL
LIN {X 0,Y 405.417,Z 420.525,A -85,B 0,C 180,E1 -17816.04,E2 -17816.04} C_VEL
LIN {X 0,Y 404.701,Z 417.737,A -85,B 0,C 180,E1 -17819.717,E2 -17819.717} C_VEL
LIN {X 0,Y 404.736,Z 418.235,A -85,B 0,C 180,E1 -17821.557,E2 -17821.557} C_VEL
LIN {X 0,Y 408.462,Z 423.69,A -85,B 0,C 180,E1 -17828.73,E2 -17828.73} C_VEL
LIN {X 0,Y 409.64,Z 424.377,A -85,B 0,C 180,E1 -17829.838,E2 -17829.838} C_VEL
LIN {X 0,Y 411.764,Z 428.108,A -85,B 0,C 180,E1 -17831.77,E2 -17831.77} C_VEL
LIN {X 0,Y 414.712,Z 430.765,A -85,B 0,C 180,E1 -17833.81,E2 -17833.81} C_VEL
LIN {X 0,Y 417.727,Z 434.98,A -85,B 0,C 180,E1 -17835.693,E2 -17835.693} C_VEL
LIN {X 0,Y 419.639,Z 436.878,A -85,B 0,C 180,E1 -17836.721,E2 -17836.721} C_VEL
LIN {X 0,Y 423.364,Z 441.554,A -85,B 0,C 180,E1 -17838.593,E2 -17838.593} C_VEL
LIN {X 0,Y 428.986,Z 448.857,A -85,B 0,C 180,E1 -17841.071,E2 -17841.071} C_VEL
LIN {X 0,Y 433.415,Z 454.657,A -85,B 0,C 180,E1 -17842.804,E2 -17842.804} C_VEL
LIN {X 0,Y 439.993,Z 463.33,A -85,B 0,C 180,E1 -17845.112,E2 -17845.112} C_VEL
LIN {X 0,Y 448.397,Z 475.294,A -85,B 0,C 180,E1 -17847.742,E2 -17847.742} C_VEL
LIN {X 0,Y 456.459,Z 487.305,A -85,B 0,C 180,E1 -17850,E2 -17850} C_VEL
LIN {X 0,Y 465.494,Z 501.628,A -85,B 0,C 180,E1 -17852.298,E2 -17852.298} C_VEL
LIN {X 0,Y 465.972,Z 502.849,A -85,B 0,C 180,E1 -17852.426,E2 -17852.426} C_VEL
LIN {X 0,Y 451.164,Z 741.354,A -85,B 0,C 180,E1 -17856.261,E2 -17856.261} C_VEL
LIN {X 0,Y 448.807,Z 765.345,A -85,B 0,C 180,E1 -17856.762,E2 -17856.762} C_VEL
LIN {X 0,Y 445.346,Z 789.027,A -85,B 0,C 180,E1 -17857.448,E2 -17857.448} C_VEL
LIN {X 0,Y 441.738,Z 809.064,A -85,B 0,C 180,E1 -17858.183,E2 -17858.183} C_VEL
LIN {X 0,Y 436.594,Z 832.915,A -85,B 0,C 180,E1 -17859.278,E2 -17859.278} C_VEL
LIN {X 0,Y 431.454,Z 853.209,A -85,B 0,C 180,E1 -17860.422,E2 -17860.422} C_VEL
LIN {X 0,Y 425.142,Z 875.3,A -85,B 0,C 180,E1 -17861.908,E2 -17861.908} C_VEL
LIN {X 0,Y 418.923,Z 894.647,A -85,B 0,C 180,E1 -17863.482,E2 -17863.482} C_VEL
LIN {X 0,Y 412.046,Z 914.516,A -85,B 0,C 180,E1 -17865.371,E2 -17865.371} C_VEL
LIN {X 0,Y 404.907,Z 933.322,A -85,B 0,C 180,E1 -17867.516,E2 -17867.516} C_VEL
LIN {X 0,Y 398.506,Z 949.471,A -85,B 0,C 180,E1 -17869.658,E2 -17869.658} C_VEL
LIN {X 0,Y 391.227,Z 966.946,A -85,B 0,C 180,E1 -17872.401,E2 -17872.401} C_VEL
LIN {X 0,Y 385.26,Z 981.041,A -85,B 0,C 180,E1 -17875,E2 -17875} C_VEL
LIN {X 0,Y 378.802,Z 996.179,A -85,B 0,C 180,E1 -17878.313,E2 -17878.313} C_VEL
LIN {X 0,Y 374.056,Z 1007.537,A -85,B 0,C 180,E1 -17881.257,E2 -17881.257} C_VEL
LIN {X 0,Y 369.221,Z 1019.655,A -85,B 0,C 180,E1 -17885.01,E2 -17885.01} C_VEL
LIN {X 0,Y 365.959,Z 1028.572,A -85,B 0,C 180,E1 -17888.355,E2 -17888.355} C_VEL
LIN {X 0,Y 363.162,Z 1037.277,A -85,B 0,C 180,E1 -17892.371,E2 -17892.371} C_VEL
LIN {X 0,Y 361.616,Z 1043.064,A -85,B 0,C 180,E1 -17895.754,E2 -17895.754} C_VEL
LIN {X 0,Y 360.594,Z 1048.184,A -85,B 0,C 180,E1 -17899.616,E2 -17899.616} C_VEL
LIN {X 0,Y 360.147,Z 1051.431,A -85,B 0,C 180,E1 -17903.304,E2 -17903.304} C_VEL
LIN {X 0,Y 360.007,Z 1053.161,A -85,B 0,C 180,E1 -17906.497,E2 -17906.497} C_VEL
LIN {X 0,Y 359.977,Z 1053.892,A -85,B 0,C 180,E1 -17910.159,E2 -17910.159} C_VEL
LIN {X 0,Y 360.009,Z 1053.139,A -85,B 0,C 180,E1 -17913.663,E2 -17913.663} C_VEL
LIN {X 0,Y 360.147,Z 1051.395,A -85,B 0,C 180,E1 -17916.857,E2 -17916.857} C_VEL
LIN {X 0,Y 360.611,Z 1048.132,A -85,B 0,C 180,E1 -17920.545,E2 -17920.545} C_VEL
LIN {X 0,Y 361.646,Z 1042.978,A -85,B 0,C 180,E1 -17924.409,E2 -17924.409} C_VEL
LIN {X 0,Y 363.208,Z 1037.174,A -85,B 0,C 180,E1 -17927.793,E2 -17927.793} C_VEL
LIN {X 0,Y 366.028,Z 1028.431,A -85,B 0,C 180,E1 -17931.809,E2 -17931.809} C_VEL
LIN {X 0,Y 369.135,Z 1019.939,A -85,B 0,C 180,E1 -17934.997,E2 -17934.997} C_VEL
LIN {X 0,Y 373.97,Z 1007.832,A -85,B 0,C 180,E1 -17938.768,E2 -17938.768} C_VEL
LIN {X 0,Y 378.874,Z 996.112,A -85,B 0,C 180,E1 -17941.81,E2 -17941.81} C_VEL
LIN {X 0,Y 385.119,Z 981.515,A -85,B 0,C 180,E1 -17945.015,E2 -17945.015} C_VEL
LIN {X 0,Y 388.953,Z 972.574,A -85,B 0,C 180,E1 -17946.727,E2 -17946.727} C_VEL
LIN {X 0,Y 390.062,Z 967.961,A -85,B 0,C 180,E1 -17947.63,E2 -17947.63} C_VEL
LIN {X 0,Y 390.316,Z 956.045,A -85,B 0,C 180,E1 -17950.211,E2 -17950.211} C_VEL
LIN {X 0,Y 391.558,Z 951.733,A -85,B 0,C 180,E1 -17950.932,E2 -17950.932} C_VEL
LIN {X 0,Y 398.747,Z 934.204,A -85,B 0,C 180,E1 -17953.301,E2 -17953.301} C_VEL
LIN {X 0,Y 405.869,Z 916.098,A -85,B 0,C 180,E1 -17955.396,E2 -17955.396} C_VEL
LIN {X 0,Y 413.048,Z 896.151,A -85,B 0,C 180,E1 -17957.327,E2 -17957.327} C_VEL
LIN {X 0,Y 419.35,Z 877.167,A -85,B 0,C 180,E1 -17958.891,E2 -17958.891} C_VEL
LIN {X 0,Y 426.068,Z 854.59,A -85,B 0,C 180,E1 -17960.437,E2 -17960.437} C_VEL
LIN {X 0,Y 431.338,Z 834.439,A -85,B 0,C 180,E1 -17961.584,E2 -17961.584} C_VEL
LIN {X 0,Y 436.756,Z 810.285,A -85,B 0,C 180,E1 -17962.707,E2 -17962.707} C_VEL
LIN {X 0,Y 440.628,Z 789.376,A -85,B 0,C 180,E1 -17963.478,E2 -17963.478} C_VEL
LIN {X 0,Y 444.18,Z 765.697,A -85,B 0,C 180,E1 -17964.166,E2 -17964.166} C_VEL
LIN {X 0,Y 446.615,Z 741.552,A -85,B 0,C 180,E1 -17964.671,E2 -17964.671} C_VEL
LIN {X 0,Y 461.648,Z 506.65,A -85,B 0,C 180,E1 -17968.457,E2 -17968.457} C_VEL
LIN {X 0,Y 451.77,Z 490.976,A -85,B 0,C 180,E1 -17971.079,E2 -17971.079} C_VEL
LIN {X 0,Y 443.038,Z 477.979,A -85,B 0,C 180,E1 -17973.674,E2 -17973.674} C_VEL
LIN {X 0,Y 435.91,Z 468.019,A -85,B 0,C 180,E1 -17976.046,E2 -17976.046} C_VEL
LIN {X 0,Y 429.746,Z 459.576,A -85,B 0,C 180,E1 -17978.359,E2 -17978.359} C_VEL
LIN {X 0,Y 425.312,Z 453.87,A -85,B 0,C 180,E1 -17980.212,E2 -17980.212} C_VEL
LIN {X 0,Y 421.411,Z 448.786,A -85,B 0,C 180,E1 -17982.034,E2 -17982.034} C_VEL
LIN {X 0,Y 417.405,Z 443.649,A -85,B 0,C 180,E1 -17984.152,E2 -17984.152} C_VEL
LIN {X 0,Y 414.068,Z 439.748,A -85,B 0,C 180,E1 -17986.169,E2 -17986.169} C_VEL
LIN {X 0,Y 412.909,Z 437.928,A -85,B 0,C 180,E1 -17986.985,E2 -17986.985} C_VEL
LIN {X 0,Y 409.829,Z 434.91,A -85,B 0,C 180,E1 -17989.314,E2 -17989.314} C_VEL
LIN {X 0,Y 408.316,Z 432.004,A -85,B 0,C 180,E1 -17990.841,E2 -17990.841} C_VEL
LIN {X 0,Y 403.95,Z 426.821,A -85,B 0,C 180,E1 -17999.291,E2 -17999.291} C_VEL
LIN {X 0,Y 403.987,Z 427.05,A -85,B 0,C 180,E1 -18000.993,E2 -18000.993} C_VEL
LIN {X 0,Y 408.492,Z 432.281,A -85,B 0,C 180,E1 -18009.013,E2 -18009.013} C_VEL
LIN {X 0,Y 410.875,Z 436.198,A -85,B 0,C 180,E1 -18011.226,E2 -18011.226} C_VEL
LIN {X 0,Y 413.46,Z 438.647,A -85,B 0,C 180,E1 -18013.069,E2 -18013.069} C_VEL
LIN {X 0,Y 416.76,Z 443.049,A -85,B 0,C 180,E1 -18015.16,E2 -18015.16} C_VEL
LIN {X 0,Y 418.195,Z 444.665,A -85,B 0,C 180,E1 -18015.96,E2 -18015.96} C_VEL
LIN {X 0,Y 421.91,Z 449.294,A -85,B 0,C 180,E1 -18017.873,E2 -18017.873} C_VEL
LIN {X 0,Y 427.346,Z 456.486,A -85,B 0,C 180,E1 -18020.332,E2 -18020.332} C_VEL
LIN {X 0,Y 431.754,Z 462.576,A -85,B 0,C 180,E1 -18022.107,E2 -18022.107} C_VEL
LIN {X 0,Y 439.997,Z 475.261,A -85,B 0,C 180,E1 -18025.076,E2 -18025.076} C_VEL
LIN {X 0,Y 449.218,Z 490.504,A -85,B 0,C 180,E1 -18027.976,E2 -18027.976} C_VEL
LIN {X 0,Y 458.178,Z 506.533,A -85,B 0,C 180,E1 -18030.49,E2 -18030.49} C_VEL
LIN {X 0,Y 461.419,Z 512.869,A -85,B 0,C 180,E1 -18031.348,E2 -18031.348} C_VEL
LIN {X 0,Y 445.999,Z 755.217,A -85,B 0,C 180,E1 -18035.259,E2 -18035.259} C_VEL
LIN {X 0,Y 443.461,Z 779.713,A -85,B 0,C 180,E1 -18035.758,E2 -18035.758} C_VEL
LIN {X 0,Y 439.607,Z 804.086,A -85,B 0,C 180,E1 -18036.434,E2 -18036.434} C_VEL
LIN {X 0,Y 435.087,Z 827.469,A -85,B 0,C 180,E1 -18037.276,E2 -18037.276} C_VEL
LIN {X 0,Y 429.625,Z 850.494,A -85,B 0,C 180,E1 -18038.342,E2 -18038.342} C_VEL
LIN {X 0,Y 424.235,Z 870.617,A -85,B 0,C 180,E1 -18039.476,E2 -18039.476} C_VEL
LIN {X 0,Y 417.167,Z 893.722,A -85,B 0,C 180,E1 -18041.052,E2 -18041.052} C_VEL
LIN {X 0,Y 410.958,Z 912.192,A -85,B 0,C 180,E1 -18042.563,E2 -18042.563} C_VEL
LIN {X 0,Y 403.203,Z 933.428,A -85,B 0,C 180,E1 -18044.625,E2 -18044.625} C_VEL
LIN {X 0,Y 396.657,Z 950.149,A -85,B 0,C 180,E1 -18046.551,E2 -18046.551} C_VEL
LIN {X 0,Y 389.487,Z 967.794,A -85,B 0,C 180,E1 -18048.913,E2 -18048.913} C_VEL
LIN {X 0,Y 382.51,Z 984.138,A -85,B 0,C 180,E1 -18051.527,E2 -18051.527} C_VEL
LIN {X 0,Y 375.986,Z 999.446,A -85,B 0,C 180,E1 -18054.38,E2 -18054.38} C_VEL
LIN {X 0,Y 369.728,Z 1013.981,A -85,B 0,C 180,E1 -18057.624,E2 -18057.624} C_VEL
LIN {X 0,Y 364.757,Z 1026.082,A -85,B 0,C 180,E1 -18060.794,E2 -18060.794} C_VEL
LIN {X 0,Y 360.156,Z 1037.887,A -85,B 0,C 180,E1 -18064.512,E2 -18064.512} C_VEL
LIN {X 0,Y 356.985,Z 1047.037,A -85,B 0,C 180,E1 -18067.955,E2 -18067.955} C_VEL
LIN {X 0,Y 354.444,Z 1055.638,A -85,B 0,C 180,E1 -18071.931,E2 -18071.931} C_VEL
LIN {X 0,Y 353.063,Z 1061.631,A -85,B 0,C 180,E1 -18075.401,E2 -18075.401} C_VEL
LIN {X 0,Y 352.229,Z 1066.95,A -85,B 0,C 180,E1 -18079.367,E2 -18079.367} C_VEL
LIN {X 0,Y 351.98,Z 1070.231,A -85,B 0,C 180,E1 -18082.984,E2 -18082.984} C_VEL
LIN {X 0,Y 351.953,Z 1072.013,A -85,B 0,C 180,E1 -18086.09,E2 -18086.09} C_VEL
LIN {X 0,Y 351.973,Z 1072.819,A -85,B 0,C 180,E1 -18089.349,E2 -18089.349} C_VEL
LIN {X 0,Y 351.964,Z 1072.355,A -85,B 0,C 180,E1 -18093.094,E2 -18093.094} C_VEL
LIN {X 0,Y 351.964,Z 1070.57,A -85,B 0,C 180,E1 -18096.525,E2 -18096.525} C_VEL
LIN {X 0,Y 352.146,Z 1067.722,A -85,B 0,C 180,E1 -18099.841,E2 -18099.841} C_VEL
LIN {X 0,Y 352.826,Z 1062.905,A -85,B 0,C 180,E1 -18103.771,E2 -18103.771} C_VEL
LIN {X 0,Y 354.124,Z 1056.826,A -85,B 0,C 180,E1 -18107.415,E2 -18107.415} C_VEL
LIN {X 0,Y 356.248,Z 1049.343,A -85,B 0,C 180,E1 -18111.055,E2 -18111.055} C_VEL
LIN {X 0,Y 359.48,Z 1039.705,A -85,B 0,C 180,E1 -18114.835,E2 -18114.835} C_VEL
LIN {X 0,Y 363.221,Z 1029.813,A -85,B 0,C 180,E1 -18118.082,E2 -18118.082} C_VEL
LIN {X 0,Y 368.654,Z 1016.481,A -85,B 0,C 180,E1 -18121.748,E2 -18121.748} C_VEL
LIN {X 0,Y 374.068,Z 1003.681,A -85,B 0,C 180,E1 -18124.705,E2 -18124.705} C_VEL
LIN {X 0,Y 381.06,Z 987.444,A -85,B 0,C 180,E1 -18127.88,E2 -18127.88} C_VEL
LIN {X 0,Y 387.459,Z 972.347,A -85,B 0,C 180,E1 -18130.371,E2 -18130.371} C_VEL
LIN {X 0,Y 394.961,Z 954.261,A -85,B 0,C 180,E1 -18132.922,E2 -18132.922} C_VEL
LIN {X 0,Y 401.753,Z 936.927,A -85,B 0,C 180,E1 -18134.977,E2 -18134.977} C_VEL
LIN {X 0,Y 409.058,Z 917.406,A -85,B 0,C 180,E1 -18136.959,E2 -18136.959} C_VEL
LIN {X 0,Y 416.001,Z 896.941,A -85,B 0,C 180,E1 -18138.687,E2 -18138.687} C_VEL
LIN {X 0,Y 422.251,Z 877.036,A -85,B 0,C 180,E1 -18140.106,E2 -18140.106} C_VEL
LIN {X 0,Y 428.711,Z 853.602,A -85,B 0,C 180,E1 -18141.484,E2 -18141.484} C_VEL
LIN {X 0,Y 433.884,Z 832.164,A -85,B 0,C 180,E1 -18142.51,E2 -18142.51} C_VEL
LIN {X 0,Y 438.999,Z 806.795,A -85,B 0,C 180,E1 -18143.467,E2 -18143.467} C_VEL
LIN {X 0,Y 442.562,Z 784.87,A -85,B 0,C 180,E1 -18144.099,E2 -18144.099} C_VEL
LIN {X 0,Y 445.639,Z 758.07,A -85,B 0,C 180,E1 -18144.677,E2 -18144.677} C_VEL
LIN {X 0,Y 460.083,Z 530.984,A -85,B 0,C 180,E1 -18148.353,E2 -18148.353} C_VEL
LIN {X 0,Y 461.182,Z 512.294,A -85,B 0,C 180,E1 -18148.675,E2 -18148.675} C_VEL
LIN {X 0,Y 452.898,Z 497.114,A -85,B 0,C 180,E1 -18150.905,E2 -18150.905} C_VEL
LIN {X 0,Y 444.854,Z 483.299,A -85,B 0,C 180,E1 -18153.286,E2 -18153.286} C_VEL
LIN {X 0,Y 437.22,Z 471.081,A -85,B 0,C 180,E1 -18155.799,E2 -18155.799} C_VEL
LIN {X 0,Y 429.64,Z 459.535,A -85,B 0,C 180,E1 -18158.64,E2 -18158.64} C_VEL
LIN {X 0,Y 425.191,Z 453.771,A -85,B 0,C 180,E1 -18160.492,E2 -18160.492} C_VEL
LIN {X 0,Y 421.404,Z 448.852,A -85,B 0,C 180,E1 -18162.248,E2 -18162.248} C_VEL
LIN {X 0,Y 417.795,Z 444.073,A -85,B 0,C 180,E1 -18164.131,E2 -18164.131} C_VEL
LIN {X 0,Y 413.894,Z 439.521,A -85,B 0,C 180,E1 -18166.448,E2 -18166.448} C_VEL
LIN {X 0,Y 412.916,Z 437.994,A -85,B 0,C 180,E1 -18167.127,E2 -18167.127} C_VEL
LIN {X 0,Y 409.624,Z 434.628,A -85,B 0,C 180,E1 -18169.593,E2 -18169.593} C_VEL
LIN {X 0,Y 408.219,Z 431.996,A -85,B 0,C 180,E1 -18170.981,E2 -18170.981} C_VEL
LIN {X 0,Y 404.38,Z 428.403,A -85,B 0,C 180,E1 -18176.172,E2 -18176.172} C_VEL
LIN {X 0,Y 403.72,Z 425.664,A -85,B 0,C 180,E1 -18179.858,E2 -18179.858} C_VEL
LIN {X 0,Y 403.747,Z 426.114,A -85,B 0,C 180,E1 -18181.419,E2 -18181.419} C_VEL
LIN {X 0,Y 407.357,Z 431.577,A -85,B 0,C 180,E1 -18188.611,E2 -18188.611} C_VEL
LIN {X 0,Y 408.438,Z 432.256,A -85,B 0,C 180,E1 -18189.654,E2 -18189.654} C_VEL
LIN {X 0,Y 410.615,Z 436.008,A -85,B 0,C 180,E1 -18191.661,E2 -18191.661} C_VEL
LIN {X 0,Y 413.323,Z 438.503,A -85,B 0,C 180,E1 -18193.572,E2 -18193.572} C_VEL
LIN {X 0,Y 416.406,Z 442.787,A -85,B 0,C 180,E1 -18195.53,E2 -18195.53} C_VEL
LIN {X 0,Y 418.137,Z 444.595,A -85,B 0,C 180,E1 -18196.482,E2 -18196.482} C_VEL
LIN {X 0,Y 421.983,Z 449.371,A -85,B 0,C 180,E1 -18198.441,E2 -18198.441} C_VEL
LIN {X 0,Y 427.306,Z 456.557,A -85,B 0,C 180,E1 -18200.835,E2 -18200.835} C_VEL
LIN {X 0,Y 431.435,Z 462.031,A -85,B 0,C 180,E1 -18202.483,E2 -18202.483} C_VEL
LIN {X 0,Y 437.733,Z 470.485,A -85,B 0,C 180,E1 -18204.746,E2 -18204.746} C_VEL
LIN {X 0,Y 446.908,Z 483.691,A -85,B 0,C 180,E1 -18207.662,E2 -18207.662} C_VEL
LIN {X 0,Y 456.845,Z 498.986,A -85,B 0,C 180,E1 -18210.443,E2 -18210.443} C_VEL
LIN {X 0,Y 461.48,Z 506.862,A -85,B 0,C 180,E1 -18211.647,E2 -18211.647} C_VEL
LIN {X 0,Y 446.416,Z 742.363,A -85,B 0,C 180,E1 -18215.446,E2 -18215.446} C_VEL
LIN {X 0,Y 443.896,Z 766.878,A -85,B 0,C 180,E1 -18215.967,E2 -18215.967} C_VEL
LIN {X 0,Y 440.395,Z 789.968,A -85,B 0,C 180,E1 -18216.644,E2 -18216.644} C_VEL
LIN {X 0,Y 436.39,Z 811.535,A -85,B 0,C 180,E1 -18217.446,E2 -18217.446} C_VEL
LIN {X 0,Y 431.26,Z 834.263,A -85,B 0,C 180,E1 -18218.51,E2 -18218.51} C_VEL
LIN {X 0,Y 425.995,Z 854.431,A -85,B 0,C 180,E1 -18219.657,E2 -18219.657} C_VEL
LIN {X 0,Y 419.287,Z 877.024,A -85,B 0,C 180,E1 -18221.203,E2 -18221.203} C_VEL
LIN {X 0,Y 413.131,Z 895.599,A -85,B 0,C 180,E1 -18222.731,E2 -18222.731} C_VEL
LIN {X 0,Y 406.058,Z 915.372,A -85,B 0,C 180,E1 -18224.631,E2 -18224.631} C_VEL
LIN {X 0,Y 398.704,Z 934.094,A -85,B 0,C 180,E1 -18226.793,E2 -18226.793} C_VEL
LIN {X 0,Y 391.499,Z 951.7,A -85,B 0,C 180,E1 -18229.17,E2 -18229.17} C_VEL
LIN {X 0,Y 384.496,Z 967.777,A -85,B 0,C 180,E1 -18231.763,E2 -18231.763} C_VEL
LIN {X 0,Y 378.236,Z 982.025,A -85,B 0,C 180,E1 -18234.438,E2 -18234.438} C_VEL
LIN {X 0,Y 371.832,Z 996.4,A -85,B 0,C 180,E1 -18237.648,E2 -18237.648} C_VEL
LIN {X 0,Y 366.894,Z 1007.701,A -85,B 0,C 180,E1 -18240.623,E2 -18240.623} C_VEL
LIN {X 0,Y 361.797,Z 1019.875,A -85,B 0,C 180,E1 -18244.461,E2 -18244.461} C_VEL
LIN {X 0,Y 358.345,Z 1028.807,A -85,B 0,C 180,E1 -18247.878,E2 -18247.878} C_VEL
LIN {X 0,Y 355.378,Z 1037.527,A -85,B 0,C 180,E1 -18251.989,E2 -18251.989} C_VEL
LIN {X 0,Y 353.742,Z 1043.282,A -85,B 0,C 180,E1 -18255.43,E2 -18255.43} C_VEL
LIN {X 0,Y 352.642,Z 1048.401,A -85,B 0,C 180,E1 -18259.38,E2 -18259.38} C_VEL
LIN {X 0,Y 352.163,Z 1051.646,A -85,B 0,C 180,E1 -18263.151,E2 -18263.151} C_VEL
LIN {X 0,Y 352.013,Z 1053.375,A -85,B 0,C 180,E1 -18266.417,E2 -18266.417} C_VEL
LIN {X 0,Y 351.98,Z 1054.106,A -85,B 0,C 180,E1 -18270.163,E2 -18270.163} C_VEL
LIN {X 0,Y 352.016,Z 1053.352,A -85,B 0,C 180,E1 -18273.746,E2 -18273.746} C_VEL
LIN {X 0,Y 352.164,Z 1051.609,A -85,B 0,C 180,E1 -18277.013,E2 -18277.013} C_VEL
LIN {X 0,Y 352.661,Z 1048.347,A -85,B 0,C 180,E1 -18280.785,E2 -18280.785} C_VEL
LIN {X 0,Y 353.775,Z 1043.194,A -85,B 0,C 180,E1 -18284.736,E2 -18284.736} C_VEL
LIN {X 0,Y 355.439,Z 1037.391,A -85,B 0,C 180,E1 -18288.195,E2 -18288.195} C_VEL
LIN {X 0,Y 358.424,Z 1028.648,A -85,B 0,C 180,E1 -18292.296,E2 -18292.296} C_VEL
LIN {X 0,Y 361.707,Z 1020.157,A -85,B 0,C 180,E1 -18295.546,E2 -18295.546} C_VEL
LIN {X 0,Y 366.783,Z 1008.05,A -85,B 0,C 180,E1 -18299.387,E2 -18299.387} C_VEL
LIN {X 0,Y 371.704,Z 996.787,A -85,B 0,C 180,E1 -18302.365,E2 -18302.365} C_VEL
LIN {X 0,Y 378.094,Z 982.494,A -85,B 0,C 180,E1 -18305.577,E2 -18305.577} C_VEL
LIN {X 0,Y 384.338,Z 968.288,A -85,B 0,C 180,E1 -18308.256,E2 -18308.256} C_VEL
LIN {X 0,Y 391.558,Z 951.733,A -85,B 0,C 180,E1 -18310.932,E2 -18310.932} C_VEL
LIN {X 0,Y 392.92,Z 946.679,A -85,B 0,C 180,E1 -18311.763,E2 -18311.763} C_VEL
LIN {X 0,Y 393.678,Z 934.138,A -85,B 0,C 180,E1 -18314.054,E2 -18314.054} C_VEL
LIN {X 0,Y 395.255,Z 928.695,A -85,B 0,C 180,E1 -18314.832,E2 -18314.832} C_VEL
LIN {X 0,Y 402.652,Z 909.777,A -85,B 0,C 180,E1 -18316.893,E2 -18316.893} C_VEL
LIN {X 0,Y 409.299,Z 891.569,A -85,B 0,C 180,E1 -18318.589,E2 -18318.589} C_VEL
LIN {X 0,Y 416.515,Z 869.655,A -85,B 0,C 180,E1 -18320.3,E2 -18320.3} C_VEL
LIN {X 0,Y 422.383,Z 849.798,A -85,B 0,C 180,E1 -18321.588,E2 -18321.588} C_VEL
LIN {X 0,Y 428.692,Z 825.074,A -85,B 0,C 180,E1 -18322.91,E2 -18322.91} C_VEL
LIN {X 0,Y 433.074,Z 804.738,A -85,B 0,C 180,E1 -18323.786,E2 -18323.786} C_VEL
LIN {X 0,Y 437.478,Z 779.985,A -85,B 0,C 180,E1 -18324.632,E2 -18324.632} C_VEL
LIN {X 0,Y 440.51,Z 757.227,A -85,B 0,C 180,E1 -18325.211,E2 -18325.211} C_VEL
LIN {X 0,Y 442.837,Z 731.393,A -85,B 0,C 180,E1 -18325.698,E2 -18325.698} C_VEL
LIN {X 0,Y 457.212,Z 510.862,A -85,B 0,C 180,E1 -18329.253,E2 -18329.253} C_VEL
LIN {X 0,Y 448.102,Z 496.31,A -85,B 0,C 180,E1 -18331.767,E2 -18331.767} C_VEL
LIN {X 0,Y 439.874,Z 483.931,A -85,B 0,C 180,E1 -18334.304,E2 -18334.304} C_VEL
LIN {X 0,Y 433.449,Z 474.805,A -85,B 0,C 180,E1 -18336.515,E2 -18336.515} C_VEL
LIN {X 0,Y 427.497,Z 466.577,A -85,B 0,C 180,E1 -18338.816,E2 -18338.816} C_VEL
LIN {X 0,Y 423.314,Z 461.078,A -85,B 0,C 180,E1 -18340.618,E2 -18340.618} C_VEL
LIN {X 0,Y 419.77,Z 456.339,A -85,B 0,C 180,E1 -18342.32,E2 -18342.32} C_VEL
LIN {X 0,Y 415.837,Z 451.253,A -85,B 0,C 180,E1 -18344.448,E2 -18344.448} C_VEL
LIN {X 0,Y 412.489,Z 447.124,A -85,B 0,C 180,E1 -18346.543,E2 -18346.543} C_VEL
LIN {X 0,Y 411.541,Z 445.678,A -85,B 0,C 180,E1 -18347.227,E2 -18347.227} C_VEL
LIN {X 0,Y 408.465,Z 442.479,A -85,B 0,C 180,E1 -18349.635,E2 -18349.635} C_VEL
LIN {X 0,Y 407.203,Z 439.902,A -85,B 0,C 180,E1 -18350.958,E2 -18350.958} C_VEL
LIN {X 0,Y 402.975,Z 434.763,A -85,B 0,C 180,E1 -18359.289,E2 -18359.289} C_VEL
LIN {X 0,Y 403.01,Z 435.003,A -85,B 0,C 180,E1 -18360.995,E2 -18360.995} C_VEL
LIN {X 0,Y 407.302,Z 440.134,A -85,B 0,C 180,E1 -18368.826,E2 -18368.826} C_VEL
LIN {X 0,Y 409.728,Z 444.094,A -85,B 0,C 180,E1 -18371.116,E2 -18371.116} C_VEL
LIN {X 0,Y 412.083,Z 446.37,A -85,B 0,C 180,E1 -18372.828,E2 -18372.828} C_VEL
LIN {X 0,Y 415.44,Z 450.852,A -85,B 0,C 180,E1 -18374.995,E2 -18374.995} C_VEL
LIN {X 0,Y 416.728,Z 452.412,A -85,B 0,C 180,E1 -18375.732,E2 -18375.732} C_VEL
LIN {X 0,Y 421.245,Z 458.319,A -85,B 0,C 180,E1 -18378.081,E2 -18378.081} C_VEL
LIN {X 0,Y 425.455,Z 463.849,A -85,B 0,C 180,E1 -18379.996,E2 -18379.996} C_VEL
LIN {X 0,Y 429.702,Z 469.858,A -85,B 0,C 180,E1 -18381.751,E2 -18381.751} C_VEL
LIN {X 0,Y 437.715,Z 482.444,A -85,B 0,C 180,E1 -18384.711,E2 -18384.711} C_VEL
LIN {X 0,Y 446.496,Z 497.239,A -85,B 0,C 180,E1 -18387.545,E2 -18387.545} C_VEL
LIN {X 0,Y 455.388,Z 513.459,A -85,B 0,C 180,E1 -18390.106,E2 -18390.106} C_VEL
LIN {X 0,Y 457.008,Z 516.883,A -85,B 0,C 180,E1 -18390.555,E2 -18390.555} C_VEL
LIN {X 0,Y 441.342,Z 755.881,A -85,B 0,C 180,E1 -18394.424,E2 -18394.424} C_VEL
LIN {X 0,Y 438.635,Z 780.767,A -85,B 0,C 180,E1 -18394.937,E2 -18394.937} C_VEL
LIN {X 0,Y 434.761,Z 804.521,A -85,B 0,C 180,E1 -18395.602,E2 -18395.602} C_VEL
LIN {X 0,Y 430.098,Z 827.985,A -85,B 0,C 180,E1 -18396.449,E2 -18396.449} C_VEL
LIN {X 0,Y 424.464,Z 851.004,A -85,B 0,C 180,E1 -18397.523,E2 -18397.523} C_VEL
LIN {X 0,Y 418.656,Z 872.054,A -85,B 0,C 180,E1 -18398.718,E2 -18398.718} C_VEL
LIN {X 0,Y 411.62,Z 894.231,A -85,B 0,C 180,E1 -18400.253,E2 -18400.253} C_VEL
LIN {X 0,Y 405.201,Z 912.748,A -85,B 0,C 180,E1 -18401.78,E2 -18401.78} C_VEL
LIN {X 0,Y 396.99,Z 934.437,A -85,B 0,C 180,E1 -18403.917,E2 -18403.917} C_VEL
LIN {X 0,Y 390.123,Z 951.4,A -85,B 0,C 180,E1 -18405.904,E2 -18405.904} C_VEL
LIN {X 0,Y 382.038,Z 970.383,A -85,B 0,C 180,E1 -18408.535,E2 -18408.535} C_VEL
LIN {X 0,Y 375.311,Z 985.628,A -85,B 0,C 180,E1 -18411.043,E2 -18411.043} C_VEL
LIN {X 0,Y 368.278,Z 1001.422,A -85,B 0,C 180,E1 -18414.095,E2 -18414.095} C_VEL
LIN {X 0,Y 362.463,Z 1014.404,A -85,B 0,C 180,E1 -18417.081,E2 -18417.081} C_VEL
LIN {X 0,Y 357.075,Z 1027.021,A -85,B 0,C 180,E1 -18420.472,E2 -18420.472} C_VEL
LIN {X 0,Y 352.514,Z 1038.134,A -85,B 0,C 180,E1 -18424.099,E2 -18424.099} C_VEL
LIN {X 0,Y 349.077,Z 1047.642,A -85,B 0,C 180,E1 -18427.784,E2 -18427.784} C_VEL
LIN {X 0,Y 346.558,Z 1055.711,A -85,B 0,C 180,E1 -18431.67,E2 -18431.67} C_VEL
LIN {X 0,Y 345.108,Z 1061.674,A -85,B 0,C 180,E1 -18435.228,E2 -18435.228} C_VEL
LIN {X 0,Y 344.216,Z 1067.063,A -85,B 0,C 180,E1 -18439.455,E2 -18439.455} C_VEL
LIN {X 0,Y 343.981,Z 1070.134,A -85,B 0,C 180,E1 -18442.987,E2 -18442.987} C_VEL
LIN {X 0,Y 343.956,Z 1071.869,A -85,B 0,C 180,E1 -18446.166,E2 -18446.166} C_VEL
LIN {X 0,Y 343.976,Z 1072.652,A -85,B 0,C 180,E1 -18449.667,E2 -18449.667} C_VEL
LIN {X 0,Y 343.961,Z 1072.002,A -85,B 0,C 180,E1 -18453.5,E2 -18453.5} C_VEL
LIN {X 0,Y 343.966,Z 1070.355,A -85,B 0,C 180,E1 -18456.677,E2 -18456.677} C_VEL
LIN {X 0,Y 344.165,Z 1067.538,A -85,B 0,C 180,E1 -18460.039,E2 -18460.039} C_VEL
LIN {X 0,Y 344.908,Z 1062.687,A -85,B 0,C 180,E1 -18464.094,E2 -18464.094} C_VEL
LIN {X 0,Y 346.3,Z 1056.606,A -85,B 0,C 180,E1 -18467.822,E2 -18467.822} C_VEL
LIN {X 0,Y 348.56,Z 1049.122,A -85,B 0,C 180,E1 -18471.542,E2 -18471.542} C_VEL
LIN {X 0,Y 351.983,Z 1039.483,A -85,B 0,C 180,E1 -18475.401,E2 -18475.401} C_VEL
LIN {X 0,Y 355.926,Z 1029.59,A -85,B 0,C 180,E1 -18478.71,E2 -18478.71} C_VEL
LIN {X 0,Y 361.818,Z 1015.796,A -85,B 0,C 180,E1 -18482.555,E2 -18482.555} C_VEL
LIN {X 0,Y 367.282,Z 1003.458,A -85,B 0,C 180,E1 -18485.441,E2 -18485.441} C_VEL
LIN {X 0,Y 374.557,Z 987.221,A -85,B 0,C 180,E1 -18488.658,E2 -18488.658} C_VEL
LIN {X 0,Y 381.2,Z 972.124,A -85,B 0,C 180,E1 -18491.176,E2 -18491.176} C_VEL
LIN {X 0,Y 388.988,Z 953.991,A -85,B 0,C 180,E1 -18493.754,E2 -18493.754} C_VEL
LIN {X 0,Y 396.208,Z 936.152,A -85,B 0,C 180,E1 -18495.877,E2 -18495.877} C_VEL
LIN {X 0,Y 403.753,Z 916.567,A -85,B 0,C 180,E1 -18497.866,E2 -18497.866} C_VEL
LIN {X 0,Y 410.941,Z 895.903,A -85,B 0,C 180,E1 -18499.604,E2 -18499.604} C_VEL
LIN {X 0,Y 417.663,Z 875.005,A -85,B 0,C 180,E1 -18501.082,E2 -18501.082} C_VEL
LIN {X 0,Y 423.73,Z 853.328,A -85,B 0,C 180,E1 -18502.343,E2 -18502.343} C_VEL
LIN {X 0,Y 428.827,Z 832.737,A -85,B 0,C 180,E1 -18503.331,E2 -18503.331} C_VEL
LIN {X 0,Y 434.197,Z 806.896,A -85,B 0,C 180,E1 -18504.31,E2 -18504.31} C_VEL
LIN {X 0,Y 437.838,Z 785.035,A -85,B 0,C 180,E1 -18504.941,E2 -18504.941} C_VEL
LIN {X 0,Y 441.024,Z 758.05,A -85,B 0,C 180,E1 -18505.525,E2 -18505.525} C_VEL
LIN {X 0,Y 455.791,Z 532.61,A -85,B 0,C 180,E1 -18509.183,E2 -18509.183} C_VEL
LIN {X 0,Y 456.807,Z 516.323,A -85,B 0,C 180,E1 -18509.459,E2 -18509.459} C_VEL
LIN {X 0,Y 448.998,Z 501.885,A -85,B 0,C 180,E1 -18511.647,E2 -18511.647} C_VEL
LIN {X 0,Y 441.827,Z 489.418,A -85,B 0,C 180,E1 -18513.849,E2 -18513.849} C_VEL
LIN {X 0,Y 434.721,Z 477.841,A -85,B 0,C 180,E1 -18516.264,E2 -18516.264} C_VEL
LIN {X 0,Y 427.471,Z 466.557,A -85,B 0,C 180,E1 -18519.066,E2 -18519.066} C_VEL
LIN {X 0,Y 423.333,Z 461.146,A -85,B 0,C 180,E1 -18520.834,E2 -18520.834} C_VEL
LIN {X 0,Y 419.62,Z 456.269,A -85,B 0,C 180,E1 -18522.6,E2 -18522.6} C_VEL
LIN {X 0,Y 415.67,Z 451.114,A -85,B 0,C 180,E1 -18524.728,E2 -18524.728} C_VEL
LIN {X 0,Y 412.119,Z 446.554,A -85,B 0,C 180,E1 -18526.96,E2 -18526.96} C_VEL
LIN {X 0,Y 411.135,Z 445.448,A -85,B 0,C 180,E1 -18527.642,E2 -18527.642} C_VEL
LIN {X 0,Y 407.892,Z 441.568,A -85,B 0,C 180,E1 -18530.262,E2 -18530.262} C_VEL
LIN {X 0,Y 406.954,Z 439.818,A -85,B 0,C 180,E1 -18531.238,E2 -18531.238} C_VEL
LIN {X 0,Y 403.247,Z 436.017,A -85,B 0,C 180,E1 -18536.588,E2 -18536.588} C_VEL
LIN {X 0,Y 402.744,Z 433.61,A -85,B 0,C 180,E1 -18539.858,E2 -18539.858} C_VEL
LIN {X 0,Y 402.765,Z 434.111,A -85,B 0,C 180,E1 -18541.423,E2 -18541.423} C_VEL
LIN {X 0,Y 406.391,Z 439.54,A -85,B 0,C 180,E1 -18548.632,E2 -18548.632} C_VEL
LIN {X 0,Y 407.242,Z 440.121,A -85,B 0,C 180,E1 -18549.468,E2 -18549.468} C_VEL
LIN {X 0,Y 409.467,Z 443.905,A -85,B 0,C 180,E1 -18551.551,E2 -18551.551} C_VEL
LIN {X 0,Y 411.942,Z 446.234,A -85,B 0,C 180,E1 -18553.332,E2 -18553.332} C_VEL
LIN {X 0,Y 415.088,Z 450.592,A -85,B 0,C 180,E1 -18555.366,E2 -18555.366} C_VEL
LIN {X 0,Y 416.634,Z 452.289,A -85,B 0,C 180,E1 -18556.236,E2 -18556.236} C_VEL
LIN {X 0,Y 421.111,Z 458.206,A -85,B 0,C 180,E1 -18558.552,E2 -18558.552} C_VEL
LIN {X 0,Y 425.485,Z 464.03,A -85,B 0,C 180,E1 -18560.533,E2 -18560.533} C_VEL
LIN {X 0,Y 429.791,Z 469.857,A -85,B 0,C 180,E1 -18562.285,E2 -18562.285} C_VEL
LIN {X 0,Y 436.017,Z 478.448,A -85,B 0,C 180,E1 -18564.56,E2 -18564.56} C_VEL
LIN {X 0,Y 444.422,Z 490.737,A -85,B 0,C 180,E1 -18567.285,E2 -18567.285} C_VEL
LIN {X 0,Y 453.897,Z 505.561,A -85,B 0,C 180,E1 -18570.004,E2 -18570.004} C_VEL
LIN {X 0,Y 457.062,Z 511.08,A -85,B 0,C 180,E1 -18570.857,E2 -18570.857} C_VEL
LIN {X 0,Y 441.743,Z 743.592,A -85,B 0,C 180,E1 -18574.619,E2 -18574.619} C_VEL
LIN {X 0,Y 439.015,Z 768.616,A -85,B 0,C 180,E1 -18575.161,E2 -18575.161} C_VEL
LIN {X 0,Y 435.59,Z 790.579,A -85,B 0,C 180,E1 -18575.811,E2 -18575.811} C_VEL
LIN {X 0,Y 431.409,Z 812.496,A -85,B 0,C 180,E1 -18576.629,E2 -18576.629} C_VEL
LIN {X 0,Y 426.006,Z 835.611,A -85,B 0,C 180,E1 -18577.723,E2 -18577.723} C_VEL
LIN {X 0,Y 420.624,Z 855.619,A -85,B 0,C 180,E1 -18578.871,E2 -18578.871} C_VEL
LIN {X 0,Y 413.463,Z 878.859,A -85,B 0,C 180,E1 -18580.486,E2 -18580.486} C_VEL
LIN {X 0,Y 407.124,Z 897.371,A -85,B 0,C 180,E1 -18582.031,E2 -18582.031} C_VEL
LIN {X 0,Y 399.15,Z 918.636,A -85,B 0,C 180,E1 -18584.139,E2 -18584.139} C_VEL
LIN {X 0,Y 392.342,Z 935.416,A -85,B 0,C 180,E1 -18586.117,E2 -18586.117} C_VEL
LIN {X 0,Y 384.924,Z 952.859,A -85,B 0,C 180,E1 -18588.517,E2 -18588.517} C_VEL
LIN {X 0,Y 377.712,Z 968.836,A -85,B 0,C 180,E1 -18591.142,E2 -18591.142} C_VEL
LIN {X 0,Y 370.916,Z 983.77,A -85,B 0,C 180,E1 -18594.008,E2 -18594.008} C_VEL
LIN {X 0,Y 364.62,Z 997.249,A -85,B 0,C 180,E1 -18597.114,E2 -18597.114} C_VEL
LIN {X 0,Y 359.26,Z 1009.054,A -85,B 0,C 180,E1 -18600.304,E2 -18600.304} C_VEL
LIN {X 0,Y 354.208,Z 1020.547,A -85,B 0,C 180,E1 -18604.053,E2 -18604.053} C_VEL
LIN {X 0,Y 350.619,Z 1029.41,A -85,B 0,C 180,E1 -18607.534,E2 -18607.534} C_VEL
LIN {X 0,Y 347.531,Z 1038.012,A -85,B 0,C 180,E1 -18611.723,E2 -18611.723} C_VEL
LIN {X 0,Y 345.813,Z 1043.749,A -85,B 0,C 180,E1 -18615.259,E2 -18615.259} C_VEL
LIN {X 0,Y 344.633,Z 1048.928,A -85,B 0,C 180,E1 -18619.468,E2 -18619.468} C_VEL
LIN {X 0,Y 344.18,Z 1051.861,A -85,B 0,C 180,E1 -18622.992,E2 -18622.992} C_VEL
LIN {X 0,Y 344.018,Z 1053.589,A -85,B 0,C 180,E1 -18626.334,E2 -18626.334} C_VEL
LIN {X 0,Y 343.983,Z 1054.319,A -85,B 0,C 180,E1 -18630.167,E2 -18630.167} C_VEL
LIN {X 0,Y 344.022,Z 1053.566,A -85,B 0,C 180,E1 -18633.833,E2 -18633.833} C_VEL
LIN {X 0,Y 344.183,Z 1051.823,A -85,B 0,C 180,E1 -18637.176,E2 -18637.176} C_VEL
LIN {X 0,Y 344.716,Z 1048.563,A -85,B 0,C 180,E1 -18641.037,E2 -18641.037} C_VEL
LIN {X 0,Y 345.847,Z 1043.659,A -85,B 0,C 180,E1 -18644.911,E2 -18644.911} C_VEL
LIN {X 0,Y 347.583,Z 1037.905,A -85,B 0,C 180,E1 -18648.448,E2 -18648.448} C_VEL
LIN {X 0,Y 350.698,Z 1029.264,A -85,B 0,C 180,E1 -18652.638,E2 -18652.638} C_VEL
LIN {X 0,Y 354.117,Z 1020.826,A -85,B 0,C 180,E1 -18655.955,E2 -18655.955} C_VEL
LIN {X 0,Y 359.149,Z 1009.398,A -85,B 0,C 180,E1 -18659.707,E2 -18659.707} C_VEL
LIN {X 0,Y 364.561,Z 997.484,A -85,B 0,C 180,E1 -18662.936,E2 -18662.936} C_VEL
LIN {X 0,Y 371.108,Z 983.473,A -85,B 0,C 180,E1 -18666.161,E2 -18666.161} C_VEL
LIN {X 0,Y 377.937,Z 968.504,A -85,B 0,C 180,E1 -18669.026,E2 -18669.026} C_VEL
LIN {X 0,Y 385.39,Z 952.016,A -85,B 0,C 180,E1 -18671.72,E2 -18671.72} C_VEL
LIN {X 0,Y 392.919,Z 934.233,A -85,B 0,C 180,E1 -18674.141,E2 -18674.141} C_VEL
LIN {X 0,Y 395.255,Z 928.695,A -85,B 0,C 180,E1 -18674.832,E2 -18674.832} C_VEL
LIN {X 0,Y 396.85,Z 923.188,A -85,B 0,C 180,E1 -18675.59,E2 -18675.59} C_VEL
LIN {X 0,Y 398.204,Z 908.602,A -85,B 0,C 180,E1 -18677.805,E2 -18677.805} C_VEL
LIN {X 0,Y 399.679,Z 903.547,A -85,B 0,C 180,E1 -18678.388,E2 -18678.388} C_VEL
LIN {X 0,Y 406.966,Z 883.237,A -85,B 0,C 180,E1 -18680.156,E2 -18680.156} C_VEL
LIN {X 0,Y 412.83,Z 865.385,A -85,B 0,C 180,E1 -18681.473,E2 -18681.473} C_VEL
LIN {X 0,Y 419.477,Z 842.732,A -85,B 0,C 180,E1 -18682.876,E2 -18682.876} C_VEL
LIN {X 0,Y 424.495,Z 822.721,A -85,B 0,C 180,E1 -18683.894,E2 -18683.894} C_VEL
LIN {X 0,Y 429.343,Z 800.368,A -85,B 0,C 180,E1 -18684.829,E2 -18684.829} C_VEL
LIN {X 0,Y 433.472,Z 776.219,A -85,B 0,C 180,E1 -18685.607,E2 -18685.607} C_VEL
LIN {X 0,Y 436.433,Z 753.728,A -85,B 0,C 180,E1 -18686.157,E2 -18686.157} C_VEL
LIN {X 0,Y 439.106,Z 720.4,A -85,B 0,C 180,E1 -18686.744,E2 -18686.744} C_VEL
LIN {X 0,Y 452.846,Z 515.189,A -85,B 0,C 180,E1 -18690.065,E2 -18690.065} C_VEL
LIN {X 0,Y 444.212,Z 501.128,A -85,B 0,C 180,E1 -18692.556,E2 -18692.556} C_VEL
LIN {X 0,Y 435.428,Z 487.842,A -85,B 0,C 180,E1 -18695.404,E2 -18695.404} C_VEL
LIN {X 0,Y 428.235,Z 477.682,A -85,B 0,C 180,E1 -18698.063,E2 -18698.063} C_VEL
LIN {X 0,Y 422.346,Z 469.439,A -85,B 0,C 180,E1 -18700.571,E2 -18700.571} C_VEL
LIN {X 0,Y 417.877,Z 463.608,A -85,B 0,C 180,E1 -18702.74,E2 -18702.74} C_VEL
LIN {X 0,Y 414.281,Z 458.848,A -85,B 0,C 180,E1 -18704.747,E2 -18704.747} C_VEL
LIN {X 0,Y 411.019,Z 454.668,A -85,B 0,C 180,E1 -18706.852,E2 -18706.852} C_VEL
LIN {X 0,Y 410.181,Z 453.424,A -85,B 0,C 180,E1 -18707.47,E2 -18707.47} C_VEL
LIN {X 0,Y 407.115,Z 450.046,A -85,B 0,C 180,E1 -18709.957,E2 -18709.957} C_VEL
LIN {X 0,Y 405.948,Z 447.74,A -85,B 0,C 180,E1 -18711.216,E2 -18711.216} C_VEL
LIN {X 0,Y 401.994,Z 442.684,A -85,B 0,C 180,E1 -18719.43,E2 -18719.43} C_VEL
LIN {X 0,Y 402.085,Z 443.128,A -85,B 0,C 180,E1 -18721.425,E2 -18721.425} C_VEL
LIN {X 0,Y 406.177,Z 448.129,A -85,B 0,C 180,E1 -18728.708,E2 -18728.708} C_VEL
LIN {X 0,Y 408.754,Z 452.175,A -85,B 0,C 180,E1 -18731.143,E2 -18731.143} C_VEL
LIN {X 0,Y 410.713,Z 454.087,A -85,B 0,C 180,E1 -18732.585,E2 -18732.585} C_VEL
LIN {X 0,Y 414.124,Z 458.654,A -85,B 0,C 180,E1 -18734.829,E2 -18734.829} C_VEL
LIN {X 0,Y 415.611,Z 460.704,A -85,B 0,C 180,E1 -18735.703,E2 -18735.703} C_VEL
LIN {X 0,Y 419.52,Z 465.781,A -85,B 0,C 180,E1 -18737.763,E2 -18737.763} C_VEL
LIN {X 0,Y 423.797,Z 471.531,A -85,B 0,C 180,E1 -18739.754,E2 -18739.754} C_VEL
LIN {X 0,Y 427.668,Z 477.136,A -85,B 0,C 180,E1 -18741.391,E2 -18741.391} C_VEL
LIN {X 0,Y 435.364,Z 489.472,A -85,B 0,C 180,E1 -18744.31,E2 -18744.31} C_VEL
LIN {X 0,Y 443.894,Z 504.159,A -85,B 0,C 180,E1 -18747.138,E2 -18747.138} C_VEL
LIN {X 0,Y 452.598,Z 520.343,A -85,B 0,C 180,E1 -18749.71,E2 -18749.71} C_VEL
LIN {X 0,Y 444.807,Z 636.996,A -85,B 0,C 180,E1 -18751.613,E2 -18751.613} C_VEL
LIN {X 0,Y 436.564,Z 759.12,A -85,B 0,C 180,E1 -18753.616,E2 -18753.616} C_VEL
LIN {X 0,Y 433.313,Z 785.445,A -85,B 0,C 180,E1 -18754.192,E2 -18754.192} C_VEL
LIN {X 0,Y 429.56,Z 807.372,A -85,B 0,C 180,E1 -18754.827,E2 -18754.827} C_VEL
LIN {X 0,Y 424.081,Z 832.949,A -85,B 0,C 180,E1 -18755.799,E2 -18755.799} C_VEL
LIN {X 0,Y 418.863,Z 853.479,A -85,B 0,C 180,E1 -18756.785,E2 -18756.785} C_VEL
LIN {X 0,Y 412.043,Z 876.884,A -85,B 0,C 180,E1 -18758.164,E2 -18758.164} C_VEL
LIN {X 0,Y 405.452,Z 896.764,A -85,B 0,C 180,E1 -18759.587,E2 -18759.587} C_VEL
LIN {X 0,Y 397.917,Z 917.626,A -85,B 0,C 180,E1 -18761.366,E2 -18761.366} C_VEL
LIN {X 0,Y 390.334,Z 936.672,A -85,B 0,C 180,E1 -18763.323,E2 -18763.323} C_VEL
LIN {X 0,Y 382.389,Z 955.622,A -85,B 0,C 180,E1 -18765.615,E2 -18765.615} C_VEL
LIN {X 0,Y 374.611,Z 972.968,A -85,B 0,C 180,E1 -18768.142,E2 -18768.142} C_VEL
LIN {X 0,Y 367.01,Z 989.66,A -85,B 0,C 180,E1 -18770.998,E2 -18770.998} C_VEL
LIN {X 0,Y 359.905,Z 1004.746,A -85,B 0,C 180,E1 -18774.112,E2 -18774.112} C_VEL
LIN {X 0,Y 353.534,Z 1018.667,A -85,B 0,C 180,E1 -18777.495,E2 -18777.495} C_VEL
LIN {X 0,Y 348.221,Z 1030.471,A -85,B 0,C 180,E1 -18780.97,E2 -18780.97} C_VEL
LIN {X 0,Y 343.989,Z 1040.712,A -85,B 0,C 180,E1 -18784.52,E2 -18784.52} C_VEL
LIN {X 0,Y 340.406,Z 1050.332,A -85,B 0,C 180,E1 -18788.614,E2 -18788.614} C_VEL
LIN {X 0,Y 338.238,Z 1057.349,A -85,B 0,C 180,E1 -18792.273,E2 -18792.273} C_VEL
LIN {X 0,Y 336.721,Z 1063.831,A -85,B 0,C 180,E1 -18796.607,E2 -18796.607} C_VEL
LIN {X 0,Y 336.153,Z 1067.667,A -85,B 0,C 180,E1 -18800.065,E2 -18800.065} C_VEL
LIN {X 0,Y 335.965,Z 1070.386,A -85,B 0,C 180,E1 -18803.506,E2 -18803.506} C_VEL
LIN {X 0,Y 335.97,Z 1072.135,A -85,B 0,C 180,E1 -18807.441,E2 -18807.441} C_VEL
LIN {X 0,Y 335.979,Z 1072.344,A -85,B 0,C 180,E1 -18811.023,E2 -18811.023} C_VEL
LIN {X 0,Y 335.957,Z 1071.508,A -85,B 0,C 180,E1 -18814.267,E2 -18814.267} C_VEL
LIN {X 0,Y 335.994,Z 1069.672,A -85,B 0,C 180,E1 -18817.524,E2 -18817.524} C_VEL
LIN {X 0,Y 336.38,Z 1065.924,A -85,B 0,C 180,E1 -18821.661,E2 -18821.661} C_VEL
LIN {X 0,Y 337.326,Z 1060.909,A -85,B 0,C 180,E1 -18825.472,E2 -18825.472} C_VEL
LIN {X 0,Y 339.057,Z 1054.529,A -85,B 0,C 180,E1 -18829.286,E2 -18829.286} C_VEL
LIN {X 0,Y 342.026,Z 1045.725,A -85,B 0,C 180,E1 -18833.427,E2 -18833.427} C_VEL
LIN {X 0,Y 345.467,Z 1036.929,A -85,B 0,C 180,E1 -18836.841,E2 -18836.841} C_VEL
LIN {X 0,Y 350.855,Z 1024.412,A -85,B 0,C 180,E1 -18840.862,E2 -18840.862} C_VEL
LIN {X 0,Y 356.116,Z 1012.818,A -85,B 0,C 180,E1 -18843.969,E2 -18843.969} C_VEL
LIN {X 0,Y 362.965,Z 998.122,A -85,B 0,C 180,E1 -18847.304,E2 -18847.304} C_VEL
LIN {X 0,Y 369.679,Z 983.581,A -85,B 0,C 180,E1 -18850.07,E2 -18850.07} C_VEL
LIN {X 0,Y 377.282,Z 967.012,A -85,B 0,C 180,E1 -18852.767,E2 -18852.767} C_VEL
LIN {X 0,Y 384.954,Z 949.339,A -85,B 0,C 180,E1 -18855.161,E2 -18855.161} C_VEL
LIN {X 0,Y 392.353,Z 931.579,A -85,B 0,C 180,E1 -18857.218,E2 -18857.218} C_VEL
LIN {X 0,Y 400.208,Z 911.106,A -85,B 0,C 180,E1 -18859.202,E2 -18859.202} C_VEL
LIN {X 0,Y 406.562,Z 893.235,A -85,B 0,C 180,E1 -18860.667,E2 -18860.667} C_VEL
LIN {X 0,Y 414.076,Z 869.869,A -85,B 0,C 180,E1 -18862.263,E2 -18862.263} C_VEL
LIN {X 0,Y 419.531,Z 850.525,A -85,B 0,C 180,E1 -18863.352,E2 -18863.352} C_VEL
LIN {X 0,Y 425.33,Z 827.294,A -85,B 0,C 180,E1 -18864.429,E2 -18864.429} C_VEL
LIN {X 0,Y 430.049,Z 803.999,A -85,B 0,C 180,E1 -18865.266,E2 -18865.266} C_VEL
LIN {X 0,Y 434.078,Z 779.688,A -85,B 0,C 180,E1 -18865.941,E2 -18865.941} C_VEL
LIN {X 0,Y 436.761,Z 755.025,A -85,B 0,C 180,E1 -18866.444,E2 -18866.444} C_VEL
LIN {X 0,Y 452.55,Z 520.445,A -85,B 0,C 180,E1 -18870.249,E2 -18870.249} C_VEL
LIN {X 0,Y 443.632,Z 503.825,A -85,B 0,C 180,E1 -18872.88,E2 -18872.88} C_VEL
LIN {X 0,Y 434.92,Z 488.846,A -85,B 0,C 180,E1 -18875.771,E2 -18875.771} C_VEL
LIN {X 0,Y 426.547,Z 475.404,A -85,B 0,C 180,E1 -18878.982,E2 -18878.982} C_VEL
LIN {X 0,Y 421.634,Z 468.688,A -85,B 0,C 180,E1 -18881.113,E2 -18881.113} C_VEL
LIN {X 0,Y 417.852,Z 463.679,A -85,B 0,C 180,E1 -18882.954,E2 -18882.954} C_VEL
LIN {X 0,Y 414.11,Z 458.698,A -85,B 0,C 180,E1 -18885.027,E2 -18885.027} C_VEL
LIN {X 0,Y 410.65,Z 454.096,A -85,B 0,C 180,E1 -18887.27,E2 -18887.27} C_VEL
LIN {X 0,Y 406.621,Z 449.256,A -85,B 0,C 180,E1 -18890.517,E2 -18890.517} C_VEL
LIN {X 0,Y 405.842,Z 447.706,A -85,B 0,C 180,E1 -18891.356,E2 -18891.356} C_VEL
LIN {X 0,Y 402.219,Z 443.894,A -85,B 0,C 180,E1 -18896.722,E2 -18896.722} C_VEL
LIN {X 0,Y 401.765,Z 441.544,A -85,B 0,C 180,E1 -18900,E2 -18900} C_VEL
LIN {X 0,Y 401.784,Z 442.104,A -85,B 0,C 180,E1 -18901.426,E2 -18901.426} C_VEL
LIN {X 0,Y 405.287,Z 447.428,A -85,B 0,C 180,E1 -18908.513,E2 -18908.513} C_VEL
LIN {X 0,Y 406.112,Z 448.129,A -85,B 0,C 180,E1 -18909.352,E2 -18909.352} C_VEL
LIN {X 0,Y 408.495,Z 451.99,A -85,B 0,C 180,E1 -18911.579,E2 -18911.579} C_VEL
LIN {X 0,Y 410.569,Z 453.96,A -85,B 0,C 180,E1 -18913.091,E2 -18913.091} C_VEL
LIN {X 0,Y 413.773,Z 458.397,A -85,B 0,C 180,E1 -18915.2,E2 -18915.2} C_VEL
LIN {X 0,Y 415.287,Z 460.219,A -85,B 0,C 180,E1 -18916.075,E2 -18916.075} C_VEL
LIN {X 0,Y 419.449,Z 465.774,A -85,B 0,C 180,E1 -18918.269,E2 -18918.269} C_VEL
LIN {X 0,Y 423.677,Z 471.502,A -85,B 0,C 180,E1 -18920.227,E2 -18920.227} C_VEL
LIN {X 0,Y 429.636,Z 479.569,A -85,B 0,C 180,E1 -18922.654,E2 -18922.654} C_VEL
LIN {X 0,Y 437.58,Z 491.17,A -85,B 0,C 180,E1 -18925.492,E2 -18925.492} C_VEL
LIN {X 0,Y 446.074,Z 504.225,A -85,B 0,C 180,E1 -18928.154,E2 -18928.154} C_VEL
LIN {X 0,Y 452.734,Z 515.278,A -85,B 0,C 180,E1 -18930.051,E2 -18930.051} C_VEL
LIN {X 0,Y 437.176,Z 744.66,A -85,B 0,C 180,E1 -18933.771,E2 -18933.771} C_VEL
LIN {X 0,Y 434.145,Z 770.851,A -85,B 0,C 180,E1 -18934.352,E2 -18934.352} C_VEL
LIN {X 0,Y 430.775,Z 791.781,A -85,B 0,C 180,E1 -18934.979,E2 -18934.979} C_VEL
LIN {X 0,Y 426.221,Z 814.876,A -85,B 0,C 180,E1 -18935.853,E2 -18935.853} C_VEL
LIN {X 0,Y 420.834,Z 836.959,A -85,B 0,C 180,E1 -18936.916,E2 -18936.916} C_VEL
LIN {X 0,Y 414.751,Z 858.874,A -85,B 0,C 180,E1 -18938.194,E2 -18938.194} C_VEL
LIN {X 0,Y 407.978,Z 879.886,A -85,B 0,C 180,E1 -18939.685,E2 -18939.685} C_VEL
LIN {X 0,Y 401.507,Z 898.231,A -85,B 0,C 180,E1 -18941.229,E2 -18941.229} C_VEL
LIN {X 0,Y 393.285,Z 919.44,A -85,B 0,C 180,E1 -18943.354,E2 -18943.354} C_VEL
LIN {X 0,Y 386.269,Z 936.188,A -85,B 0,C 180,E1 -18945.348,E2 -18945.348} C_VEL
LIN {X 0,Y 377.964,Z 954.914,A -85,B 0,C 180,E1 -18947.987,E2 -18947.987} C_VEL
LIN {X 0,Y 370.973,Z 969.894,A -85,B 0,C 180,E1 -18950.499,E2 -18950.499} C_VEL
LIN {X 0,Y 363.603,Z 985.401,A -85,B 0,C 180,E1 -18953.56,E2 -18953.56} C_VEL
LIN {X 0,Y 357.442,Z 998.097,A -85,B 0,C 180,E1 -18956.559,E2 -18956.559} C_VEL
LIN {X 0,Y 351.638,Z 1010.406,A -85,B 0,C 180,E1 -18959.97,E2 -18959.97} C_VEL
LIN {X 0,Y 346.638,Z 1021.22,A -85,B 0,C 180,E1 -18963.627,E2 -18963.627} C_VEL
LIN {X 0,Y 342.752,Z 1030.426,A -85,B 0,C 180,E1 -18967.352,E2 -18967.352} C_VEL
LIN {X 0,Y 339.678,Z 1038.528,A -85,B 0,C 180,E1 -18971.463,E2 -18971.463} C_VEL
LIN {X 0,Y 337.886,Z 1044.216,A -85,B 0,C 180,E1 -18975.081,E2 -18975.081} C_VEL
LIN {X 0,Y 336.64,Z 1049.369,A -85,B 0,C 180,E1 -18979.465,E2 -18979.465} C_VEL
LIN {X 0,Y 336.185,Z 1052.187,A -85,B 0,C 180,E1 -18982.996,E2 -18982.996} C_VEL
LIN {X 0,Y 336.02,Z 1053.869,A -85,B 0,C 180,E1 -18986.417,E2 -18986.417} C_VEL
LIN {X 0,Y 335.981,Z 1054.51,A -85,B 0,C 180,E1 -18990.341,E2 -18990.341} C_VEL
LIN {X 0,Y 336.028,Z 1053.78,A -85,B 0,C 180,E1 -18993.924,E2 -18993.924} C_VEL
LIN {X 0,Y 336.205,Z 1052.038,A -85,B 0,C 180,E1 -18997.347,E2 -18997.347} C_VEL
LIN {X 0,Y 336.778,Z 1048.778,A -85,B 0,C 180,E1 -19001.301,E2 -19001.301} C_VEL
LIN {X 0,Y 338.022,Z 1043.756,A -85,B 0,C 180,E1 -19005.349,E2 -19005.349} C_VEL
LIN {X 0,Y 339.839,Z 1038.122,A -85,B 0,C 180,E1 -19008.884,E2 -19008.884} C_VEL
LIN {X 0,Y 343.14,Z 1029.482,A -85,B 0,C 180,E1 -19013.165,E2 -19013.165} C_VEL
LIN {X 0,Y 346.912,Z 1020.683,A -85,B 0,C 180,E1 -19016.683,E2 -19016.683} C_VEL
LIN {X 0,Y 352.288,Z 1009.05,A -85,B 0,C 180,E1 -19020.534,E2 -19020.534} C_VEL
LIN {X 0,Y 357.919,Z 997.221,A -85,B 0,C 180,E1 -19023.775,E2 -19023.775} C_VEL
LIN {X 0,Y 364.859,Z 982.927,A -85,B 0,C 180,E1 -19027.079,E2 -19027.079} C_VEL
LIN {X 0,Y 371.606,Z 968.72,A -85,B 0,C 180,E1 -19029.821,E2 -19029.821} C_VEL
LIN {X 0,Y 379.299,Z 952.279,A -85,B 0,C 180,E1 -19032.535,E2 -19032.535} C_VEL
LIN {X 0,Y 386.872,Z 934.988,A -85,B 0,C 180,E1 -19034.914,E2 -19034.914} C_VEL
LIN {X 0,Y 394.223,Z 917.44,A -85,B 0,C 180,E1 -19036.978,E2 -19036.978} C_VEL
LIN {X 0,Y 399.679,Z 903.547,A -85,B 0,C 180,E1 -19038.388,E2 -19038.388} C_VEL
LIN {X 0,Y 401.311,Z 897.592,A -85,B 0,C 180,E1 -19039.062,E2 -19039.062} C_VEL
LIN {X 0,Y 402.84,Z 881.87,A -85,B 0,C 180,E1 -19041.085,E2 -19041.085} C_VEL
LIN {X 0,Y 404.274,Z 876.455,A -85,B 0,C 180,E1 -19041.593,E2 -19041.593} C_VEL
LIN {X 0,Y 411.397,Z 854.115,A -85,B 0,C 180,E1 -19043.106,E2 -19043.106} C_VEL
LIN {X 0,Y 417.063,Z 833.907,A -85,B 0,C 180,E1 -19044.25,E2 -19044.25} C_VEL
LIN {X 0,Y 422.89,Z 809.424,A -85,B 0,C 180,E1 -19045.368,E2 -19045.368} C_VEL
LIN {X 0,Y 427.044,Z 788.337,A -85,B 0,C 180,E1 -19046.13,E2 -19046.13} C_VEL
LIN {X 0,Y 430.942,Z 762.968,A -85,B 0,C 180,E1 -19046.835,E2 -19046.835} C_VEL
LIN {X 0,Y 433.3,Z 740.628,A -85,B 0,C 180,E1 -19047.29,E2 -19047.29} C_VEL
LIN {X 0,Y 448.642,Z 519.54,A -85,B 0,C 180,E1 -19050.876,E2 -19050.876} C_VEL
LIN {X 0,Y 440.107,Z 505.644,A -85,B 0,C 180,E1 -19053.448,E2 -19053.448} C_VEL
LIN {X 0,Y 432.405,Z 493.864,A -85,B 0,C 180,E1 -19056.057,E2 -19056.057} C_VEL
LIN {X 0,Y 425.976,Z 484.611,A -85,B 0,C 180,E1 -19058.52,E2 -19058.52} C_VEL
LIN {X 0,Y 420.366,Z 476.664,A -85,B 0,C 180,E1 -19060.982,E2 -19060.982} C_VEL
LIN {X 0,Y 416.136,Z 471.011,A -85,B 0,C 180,E1 -19063.098,E2 -19063.098} C_VEL
LIN {X 0,Y 412.737,Z 466.436,A -85,B 0,C 180,E1 -19065.048,E2 -19065.048} C_VEL
LIN {X 0,Y 409.472,Z 462.043,A -85,B 0,C 180,E1 -19067.233,E2 -19067.233} C_VEL
LIN {X 0,Y 408.448,Z 460.877,A -85,B 0,C 180,E1 -19067.99,E2 -19067.99} C_VEL
LIN {X 0,Y 405.644,Z 457.355,A -85,B 0,C 180,E1 -19070.422,E2 -19070.422} C_VEL
LIN {X 0,Y 404.841,Z 455.635,A -85,B 0,C 180,E1 -19071.335,E2 -19071.335} C_VEL
LIN {X 0,Y 401.019,Z 450.626,A -85,B 0,C 180,E1 -19079.429,E2 -19079.429} C_VEL
LIN {X 0,Y 401.108,Z 451.089,A -85,B 0,C 180,E1 -19081.428,E2 -19081.428} C_VEL
LIN {X 0,Y 404.997,Z 455.967,A -85,B 0,C 180,E1 -19088.519,E2 -19088.519} C_VEL
LIN {X 0,Y 407.608,Z 460.066,A -85,B 0,C 180,E1 -19091.031,E2 -19091.031} C_VEL
LIN {X 0,Y 409.439,Z 461.97,A -85,B 0,C 180,E1 -19092.41,E2 -19092.41} C_VEL
LIN {X 0,Y 413.043,Z 466.672,A -85,B 0,C 180,E1 -19094.797,E2 -19094.797} C_VEL
LIN {X 0,Y 417.871,Z 473.342,A -85,B 0,C 180,E1 -19097.476,E2 -19097.476} C_VEL
LIN {X 0,Y 422.22,Z 479.311,A -85,B 0,C 180,E1 -19099.543,E2 -19099.543} C_VEL
LIN {X 0,Y 425.726,Z 484.543,A -85,B 0,C 180,E1 -19101.06,E2 -19101.06} C_VEL
LIN {X 0,Y 433.035,Z 496.5,A -85,B 0,C 180,E1 -19103.906,E2 -19103.906} C_VEL
LIN {X 0,Y 441.314,Z 511.076,A -85,B 0,C 180,E1 -19106.727,E2 -19106.727} C_VEL
LIN {X 0,Y 448.465,Z 524.638,A -85,B 0,C 180,E1 -19108.917,E2 -19108.917} C_VEL
LIN {X 0,Y 432.392,Z 756.351,A -85,B 0,C 180,E1 -19112.684,E2 -19112.684} C_VEL
LIN {X 0,Y 429.427,Z 781.668,A -85,B 0,C 180,E1 -19113.213,E2 -19113.213} C_VEL
LIN {X 0,Y 425.517,Z 804.53,A -85,B 0,C 180,E1 -19113.854,E2 -19113.854} C_VEL
LIN {X 0,Y 420.718,Z 827.571,A -85,B 0,C 180,E1 -19114.683,E2 -19114.683} C_VEL
LIN {X 0,Y 415.009,Z 849.867,A -85,B 0,C 180,E1 -19115.714,E2 -19115.714} C_VEL
LIN {X 0,Y 409.186,Z 869.985,A -85,B 0,C 180,E1 -19116.843,E2 -19116.843} C_VEL
LIN {X 0,Y 401.77,Z 892.473,A -85,B 0,C 180,E1 -19118.377,E2 -19118.377} C_VEL
LIN {X 0,Y 395.219,Z 910.395,A -85,B 0,C 180,E1 -19119.839,E2 -19119.839} C_VEL
LIN {X 0,Y 387.12,Z 930.945,A -85,B 0,C 180,E1 -19121.827,E2 -19121.827} C_VEL
LIN {X 0,Y 379.626,Z 948.374,A -85,B 0,C 180,E1 -19123.845,E2 -19123.845} C_VEL
LIN {X 0,Y 372.105,Z 965.116,A -85,B 0,C 180,E1 -19126.11,E2 -19126.11} C_VEL
LIN {X 0,Y 363.819,Z 982.63,A -85,B 0,C 180,E1 -19128.94,E2 -19128.94} C_VEL
LIN {X 0,Y 356.946,Z 996.886,A -85,B 0,C 180,E1 -19131.661,E2 -19131.661} C_VEL
LIN {X 0,Y 349.595,Z 1012.036,A -85,B 0,C 180,E1 -19135.108,E2 -19135.108} C_VEL
LIN {X 0,Y 344.034,Z 1023.679,A -85,B 0,C 180,E1 -19138.261,E2 -19138.261} C_VEL
LIN {X 0,Y 338.529,Z 1035.829,A -85,B 0,C 180,E1 -19142.181,E2 -19142.181} C_VEL
LIN {X 0,Y 334.613,Z 1045.142,A -85,B 0,C 180,E1 -19145.834,E2 -19145.834} C_VEL
LIN {X 0,Y 331.513,Z 1053.727,A -85,B 0,C 180,E1 -19149.889,E2 -19149.889} C_VEL
LIN {X 0,Y 329.512,Z 1060.459,A -85,B 0,C 180,E1 -19153.97,E2 -19153.97} C_VEL
LIN {X 0,Y 328.458,Z 1065.519,A -85,B 0,C 180,E1 -19157.875,E2 -19157.875} C_VEL
LIN {X 0,Y 327.998,Z 1069.411,A -85,B 0,C 180,E1 -19162.203,E2 -19162.203} C_VEL
LIN {X 0,Y 327.959,Z 1071.302,A -85,B 0,C 180,E1 -19165.628,E2 -19165.628} C_VEL
LIN {X 0,Y 327.981,Z 1072.133,A -85,B 0,C 180,E1 -19168.952,E2 -19168.952} C_VEL
LIN {X 0,Y 327.972,Z 1071.918,A -85,B 0,C 180,E1 -19172.621,E2 -19172.621} C_VEL
LIN {X 0,Y 327.967,Z 1070.158,A -85,B 0,C 180,E1 -19176.653,E2 -19176.653} C_VEL
LIN {X 0,Y 328.18,Z 1067.388,A -85,B 0,C 180,E1 -19180.227,E2 -19180.227} C_VEL
LIN {X 0,Y 328.899,Z 1063.12,A -85,B 0,C 180,E1 -19184.116,E2 -19184.116} C_VEL
LIN {X 0,Y 330.514,Z 1056.784,A -85,B 0,C 180,E1 -19188.338,E2 -19188.338} C_VEL
LIN {X 0,Y 332.846,Z 1049.76,A -85,B 0,C 180,E1 -19192.056,E2 -19192.056} C_VEL
LIN {X 0,Y 336.898,Z 1039.504,A -85,B 0,C 180,E1 -19196.435,E2 -19196.435} C_VEL
LIN {X 0,Y 341.228,Z 1029.667,A -85,B 0,C 180,E1 -19199.877,E2 -19199.877} C_VEL
LIN {X 0,Y 347.134,Z 1017.098,A -85,B 0,C 180,E1 -19203.576,E2 -19203.576} C_VEL
LIN {X 0,Y 353.21,Z 1004.429,A -85,B 0,C 180,E1 -19206.677,E2 -19206.677} C_VEL
LIN {X 0,Y 360.595,Z 989.324,A -85,B 0,C 180,E1 -19209.832,E2 -19209.832} C_VEL
LIN {X 0,Y 368.482,Z 972.611,A -85,B 0,C 180,E1 -19212.717,E2 -19212.717} C_VEL
LIN {X 0,Y 376.597,Z 955.1,A -85,B 0,C 180,E1 -19215.284,E2 -19215.284} C_VEL
LIN {X 0,Y 384.732,Z 936.259,A -85,B 0,C 180,E1 -19217.569,E2 -19217.569} C_VEL
LIN {X 0,Y 392.722,Z 916.74,A -85,B 0,C 180,E1 -19219.576,E2 -19219.576} C_VEL
LIN {X 0,Y 400.287,Z 896.274,A -85,B 0,C 180,E1 -19221.316,E2 -19221.316} C_VEL
LIN {X 0,Y 407.051,Z 876.369,A -85,B 0,C 180,E1 -19222.738,E2 -19222.738} C_VEL
LIN {X 0,Y 413.73,Z 854.016,A -85,B 0,C 180,E1 -19224.058,E2 -19224.058} C_VEL
LIN {X 0,Y 419.095,Z 833.451,A -85,B 0,C 180,E1 -19225.05,E2 -19225.05} C_VEL
LIN {X 0,Y 424.578,Z 808.729,A -85,B 0,C 180,E1 -19226,E2 -19226} C_VEL
LIN {X 0,Y 428.537,Z 786.279,A -85,B 0,C 180,E1 -19226.655,E2 -19226.655} C_VEL
LIN {X 0,Y 431.821,Z 761.229,A -85,B 0,C 180,E1 -19227.215,E2 -19227.215} C_VEL
LIN {X 0,Y 436.154,Z 700.564,A -85,B 0,C 180,E1 -19228.229,E2 -19228.229} C_VEL
LIN {X 0,Y 448.255,Z 524.445,A -85,B 0,C 180,E1 -19231.086,E2 -19231.086} C_VEL
LIN {X 0,Y 440.022,Z 508.844,A -85,B 0,C 180,E1 -19233.625,E2 -19233.625} C_VEL
LIN {X 0,Y 431.569,Z 494.129,A -85,B 0,C 180,E1 -19236.554,E2 -19236.554} C_VEL
LIN {X 0,Y 423.867,Z 481.649,A -85,B 0,C 180,E1 -19239.638,E2 -19239.638} C_VEL
LIN {X 0,Y 419.663,Z 475.892,A -85,B 0,C 180,E1 -19241.525,E2 -19241.525} C_VEL
LIN {X 0,Y 416.101,Z 471.084,A -85,B 0,C 180,E1 -19243.312,E2 -19243.312} C_VEL
LIN {X 0,Y 412.562,Z 466.279,A -85,B 0,C 180,E1 -19245.329,E2 -19245.329} C_VEL
LIN {X 0,Y 408.812,Z 461.207,A -85,B 0,C 180,E1 -19247.858,E2 -19247.858} C_VEL
LIN {X 0,Y 405.559,Z 457.327,A -85,B 0,C 180,E1 -19250.564,E2 -19250.564} C_VEL
LIN {X 0,Y 404.59,Z 455.519,A -85,B 0,C 180,E1 -19251.616,E2 -19251.616} C_VEL
LIN {X 0,Y 400.969,Z 451.111,A -85,B 0,C 180,E1 -19257.713,E2 -19257.713} C_VEL
LIN {X 0,Y 400.788,Z 449.482,A -85,B 0,C 180,E1 -19260.143,E2 -19260.143} C_VEL
LIN {X 0,Y 400.839,Z 450.417,A -85,B 0,C 180,E1 -19261.858,E2 -19261.858} C_VEL
LIN {X 0,Y 404.321,Z 455.39,A -85,B 0,C 180,E1 -19268.533,E2 -19268.533} C_VEL
LIN {X 0,Y 404.925,Z 455.975,A -85,B 0,C 180,E1 -19269.165,E2 -19269.165} C_VEL
LIN {X 0,Y 407.349,Z 459.883,A -85,B 0,C 180,E1 -19271.468,E2 -19271.468} C_VEL
LIN {X 0,Y 409.283,Z 461.838,A -85,B 0,C 180,E1 -19272.91,E2 -19272.91} C_VEL
LIN {X 0,Y 412.577,Z 466.312,A -85,B 0,C 180,E1 -19275.102,E2 -19275.102} C_VEL
LIN {X 0,Y 414.174,Z 468.492,A -85,B 0,C 180,E1 -19276.047,E2 -19276.047} C_VEL
LIN {X 0,Y 417.797,Z 473.34,A -85,B 0,C 180,E1 -19277.983,E2 -19277.983} C_VEL
LIN {X 0,Y 421.882,Z 478.973,A -85,B 0,C 180,E1 -19279.92,E2 -19279.92} C_VEL
LIN {X 0,Y 427.659,Z 486.975,A -85,B 0,C 180,E1 -19282.33,E2 -19282.33} C_VEL
LIN {X 0,Y 435.539,Z 498.667,A -85,B 0,C 180,E1 -19285.205,E2 -19285.205} C_VEL
LIN {X 0,Y 444.056,Z 512.079,A -85,B 0,C 180,E1 -19287.928,E2 -19287.928} C_VEL
LIN {X 0,Y 448.483,Z 519.672,A -85,B 0,C 180,E1 -19289.232,E2 -19289.232} C_VEL
LIN {X 0,Y 432.747,Z 745.27,A -85,B 0,C 180,E1 -19292.897,E2 -19292.897} C_VEL
LIN {X 0,Y 429.562,Z 771.827,A -85,B 0,C 180,E1 -19293.49,E2 -19293.49} C_VEL
LIN {X 0,Y 426.124,Z 792.585,A -85,B 0,C 180,E1 -19294.115,E2 -19294.115} C_VEL
LIN {X 0,Y 421.565,Z 815.099,A -85,B 0,C 180,E1 -19294.968,E2 -19294.968} C_VEL
LIN {X 0,Y 415.948,Z 837.55,A -85,B 0,C 180,E1 -19296.049,E2 -19296.049} C_VEL
LIN {X 0,Y 409.521,Z 860.089,A -85,B 0,C 180,E1 -19297.369,E2 -19297.369} C_VEL
LIN {X 0,Y 402.574,Z 880.915,A -85,B 0,C 180,E1 -19298.863,E2 -19298.863} C_VEL
LIN {X 0,Y 395.669,Z 899.913,A -85,B 0,C 180,E1 -19300.478,E2 -19300.478} C_VEL
LIN {X 0,Y 387.553,Z 920.104,A -85,B 0,C 180,E1 -19302.529,E2 -19302.529} C_VEL
LIN {X 0,Y 380.266,Z 936.961,A -85,B 0,C 180,E1 -19304.555,E2 -19304.555} C_VEL
LIN {X 0,Y 371.468,Z 956.079,A -85,B 0,C 180,E1 -19307.294,E2 -19307.294} C_VEL
LIN {X 0,Y 364.283,Z 970.952,A -85,B 0,C 180,E1 -19309.832,E2 -19309.832} C_VEL
LIN {X 0,Y 356.237,Z 987.152,A -85,B 0,C 180,E1 -19313.125,E2 -19313.125} C_VEL
LIN {X 0,Y 349.988,Z 999.573,A -85,B 0,C 180,E1 -19316.145,E2 -19316.145} C_VEL
LIN {X 0,Y 343.498,Z 1012.686,A -85,B 0,C 180,E1 -19319.955,E2 -19319.955} C_VEL
LIN {X 0,Y 338.815,Z 1022.481,A -85,B 0,C 180,E1 -19323.406,E2 -19323.406} C_VEL
LIN {X 0,Y 334.576,Z 1032.131,A -85,B 0,C 180,E1 -19327.51,E2 -19327.51} C_VEL
LIN {X 0,Y 331.726,Z 1039.341,A -85,B 0,C 180,E1 -19331.367,E2 -19331.367} C_VEL
LIN {X 0,Y 329.762,Z 1045.43,A -85,B 0,C 180,E1 -19335.424,E2 -19335.424} C_VEL
LIN {X 0,Y 328.61,Z 1049.983,A -85,B 0,C 180,E1 -19339.658,E2 -19339.658} C_VEL
LIN {X 0,Y 328.166,Z 1052.734,A -85,B 0,C 180,E1 -19343.351,E2 -19343.351} C_VEL
LIN {X 0,Y 328.002,Z 1054.423,A -85,B 0,C 180,E1 -19347.379,E2 -19347.379} C_VEL
LIN {X 0,Y 327.992,Z 1054.634,A -85,B 0,C 180,E1 -19351.048,E2 -19351.048} C_VEL
LIN {X 0,Y 328.047,Z 1053.861,A -85,B 0,C 180,E1 -19354.37,E2 -19354.37} C_VEL
LIN {X 0,Y 328.259,Z 1052.031,A -85,B 0,C 180,E1 -19357.879,E2 -19357.879} C_VEL
LIN {X 0,Y 329.017,Z 1048.213,A -85,B 0,C 180,E1 -19362.283,E2 -19362.283} C_VEL
LIN {X 0,Y 330.296,Z 1043.594,A -85,B 0,C 180,E1 -19365.991,E2 -19365.991} C_VEL
LIN {X 0,Y 332.591,Z 1037.152,A -85,B 0,C 180,E1 -19370.043,E2 -19370.043} C_VEL
LIN {X 0,Y 335.952,Z 1028.903,A -85,B 0,C 180,E1 -19374.064,E2 -19374.064} C_VEL
LIN {X 0,Y 340.066,Z 1019.907,A -85,B 0,C 180,E1 -19377.682,E2 -19377.682} C_VEL
LIN {X 0,Y 345.774,Z 1008.137,A -85,B 0,C 180,E1 -19381.561,E2 -19381.561} C_VEL
LIN {X 0,Y 351.45,Z 996.777,A -85,B 0,C 180,E1 -19384.692,E2 -19384.692} C_VEL
LIN {X 0,Y 359.081,Z 981.619,A -85,B 0,C 180,E1 -19388.183,E2 -19388.183} C_VEL
LIN {X 0,Y 365.759,Z 968.099,A -85,B 0,C 180,E1 -19390.796,E2 -19390.796} C_VEL
LIN {X 0,Y 373.998,Z 950.944,A -85,B 0,C 180,E1 -19393.612,E2 -19393.612} C_VEL
LIN {X 0,Y 381.534,Z 934.296,A -85,B 0,C 180,E1 -19395.896,E2 -19395.896} C_VEL
LIN {X 0,Y 389.634,Z 915.505,A -85,B 0,C 180,E1 -19398.091,E2 -19398.091} C_VEL
LIN {X 0,Y 397.375,Z 895.644,A -85,B 0,C 180,E1 -19400.014,E2 -19400.014} C_VEL
LIN {X 0,Y 404.274,Z 876.455,A -85,B 0,C 180,E1 -19401.593,E2 -19401.593} C_VEL
LIN {X 0,Y 405.855,Z 870.08,A -85,B 0,C 180,E1 -19402.18,E2 -19402.18} C_VEL
LIN {X 0,Y 407.368,Z 853.263,A -85,B 0,C 180,E1 -19403.993,E2 -19403.993} C_VEL
LIN {X 0,Y 408.694,Z 847.523,A -85,B 0,C 180,E1 -19404.425,E2 -19404.425} C_VEL
LIN {X 0,Y 414.594,Z 825.693,A -85,B 0,C 180,E1 -19405.57,E2 -19405.57} C_VEL
LIN {X 0,Y 419.327,Z 805.203,A -85,B 0,C 180,E1 -19406.448,E2 -19406.448} C_VEL
LIN {X 0,Y 424.053,Z 780.326,A -85,B 0,C 180,E1 -19407.29,E2 -19407.29} C_VEL
LIN {X 0,Y 427.279,Z 757.654,A -85,B 0,C 180,E1 -19407.861,E2 -19407.861} C_VEL
LIN {X 0,Y 429.805,Z 731.318,A -85,B 0,C 180,E1 -19408.355,E2 -19408.355} C_VEL
LIN {X 0,Y 444.48,Z 523.867,A -85,B 0,C 180,E1 -19411.716,E2 -19411.716} C_VEL
LIN {X 0,Y 436.108,Z 510.179,A -85,B 0,C 180,E1 -19414.357,E2 -19414.357} C_VEL
LIN {X 0,Y 428.45,Z 498.307,A -85,B 0,C 180,E1 -19417.098,E2 -19417.098} C_VEL
LIN {X 0,Y 421.522,Z 488.312,A -85,B 0,C 180,E1 -19419.947,E2 -19419.947} C_VEL
LIN {X 0,Y 417.59,Z 482.841,A -85,B 0,C 180,E1 -19421.792,E2 -19421.792} C_VEL
LIN {X 0,Y 414.535,Z 478.559,A -85,B 0,C 180,E1 -19423.391,E2 -19423.391} C_VEL
LIN {X 0,Y 411.205,Z 474.02,A -85,B 0,C 180,E1 -19425.351,E2 -19425.351} C_VEL
LIN {X 0,Y 407.944,Z 469.416,A -85,B 0,C 180,E1 -19427.616,E2 -19427.616} C_VEL
LIN {X 0,Y 404.52,Z 465.299,A -85,B 0,C 180,E1 -19430.539,E2 -19430.539} C_VEL
LIN {X 0,Y 403.599,Z 463.464,A -85,B 0,C 180,E1 -19431.595,E2 -19431.595} C_VEL
LIN {X 0,Y 400.044,Z 458.568,A -85,B 0,C 180,E1 -19439.427,E2 -19439.427} C_VEL
LIN {X 0,Y 400.129,Z 459.063,A -85,B 0,C 180,E1 -19441.432,E2 -19441.432} C_VEL
LIN {X 0,Y 403.821,Z 463.8,A -85,B 0,C 180,E1 -19448.329,E2 -19448.329} C_VEL
LIN {X 0,Y 406.464,Z 467.955,A -85,B 0,C 180,E1 -19450.919,E2 -19450.919} C_VEL
LIN {X 0,Y 408.083,Z 469.678,A -85,B 0,C 180,E1 -19452.165,E2 -19452.165} C_VEL
LIN {X 0,Y 412.263,Z 475.433,A -85,B 0,C 180,E1 -19454.969,E2 -19454.969} C_VEL
LIN {X 0,Y 416.361,Z 481.094,A -85,B 0,C 180,E1 -19457.253,E2 -19457.253} C_VEL
LIN {X 0,Y 420.371,Z 486.682,A -85,B 0,C 180,E1 -19459.202,E2 -19459.202} C_VEL
LIN {X 0,Y 423.725,Z 491.815,A -85,B 0,C 180,E1 -19460.694,E2 -19460.694} C_VEL
LIN {X 0,Y 430.728,Z 503.526,A -85,B 0,C 180,E1 -19463.497,E2 -19463.497} C_VEL
LIN {X 0,Y 438.666,Z 517.815,A -85,B 0,C 180,E1 -19466.281,E2 -19466.281} C_VEL
LIN {X 0,Y 444.319,Z 528.834,A -85,B 0,C 180,E1 -19468.081,E2 -19468.081} C_VEL
LIN {X 0,Y 428.023,Z 757.123,A -85,B 0,C 180,E1 -19471.796,E2 -19471.796} C_VEL
LIN {X 0,Y 424.715,Z 783.685,A -85,B 0,C 180,E1 -19472.364,E2 -19472.364} C_VEL
LIN {X 0,Y 420.831,Z 805.656,A -85,B 0,C 180,E1 -19472.986,E2 -19472.986} C_VEL
LIN {X 0,Y 415.513,Z 829.958,A -85,B 0,C 180,E1 -19473.88,E2 -19473.88} C_VEL
LIN {X 0,Y 410.02,Z 850.792,A -85,B 0,C 180,E1 -19474.855,E2 -19474.855} C_VEL
LIN {X 0,Y 403.786,Z 871.709,A -85,B 0,C 180,E1 -19476.039,E2 -19476.039} C_VEL
LIN {X 0,Y 396.387,Z 893.3,A -85,B 0,C 180,E1 -19477.535,E2 -19477.535} C_VEL
LIN {X 0,Y 389.75,Z 910.92,A -85,B 0,C 180,E1 -19478.983,E2 -19478.983} C_VEL
LIN {X 0,Y 381.159,Z 931.955,A -85,B 0,C 180,E1 -19481.045,E2 -19481.045} C_VEL
LIN {X 0,Y 373.56,Z 949.074,A -85,B 0,C 180,E1 -19483.053,E2 -19483.053} C_VEL
LIN {X 0,Y 365.27,Z 966.925,A -85,B 0,C 180,E1 -19485.511,E2 -19485.511} C_VEL
LIN {X 0,Y 357.199,Z 983.265,A -85,B 0,C 180,E1 -19488.224,E2 -19488.224} C_VEL
LIN {X 0,Y 349.559,Z 998.57,A -85,B 0,C 180,E1 -19491.212,E2 -19491.212} C_VEL
LIN {X 0,Y 342.273,Z 1012.891,A -85,B 0,C 180,E1 -19494.593,E2 -19494.593} C_VEL
LIN {X 0,Y 336.176,Z 1025.203,A -85,B 0,C 180,E1 -19498.033,E2 -19498.033} C_VEL
LIN {X 0,Y 330.559,Z 1037.008,A -85,B 0,C 180,E1 -19502.04,E2 -19502.04} C_VEL
LIN {X 0,Y 326.59,Z 1046.16,A -85,B 0,C 180,E1 -19505.779,E2 -19505.779} C_VEL
LIN {X 0,Y 323.237,Z 1055.056,A -85,B 0,C 180,E1 -19510.295,E2 -19510.295} C_VEL
LIN {X 0,Y 321.448,Z 1061.021,A -85,B 0,C 180,E1 -19514.113,E2 -19514.113} C_VEL
LIN {X 0,Y 320.322,Z 1066.414,A -85,B 0,C 180,E1 -19518.658,E2 -19518.658} C_VEL
LIN {X 0,Y 319.996,Z 1069.489,A -85,B 0,C 180,E1 -19522.459,E2 -19522.459} C_VEL
LIN {X 0,Y 319.96,Z 1071.228,A -85,B 0,C 180,E1 -19525.878,E2 -19525.878} C_VEL
LIN {X 0,Y 319.985,Z 1072.012,A -85,B 0,C 180,E1 -19529.642,E2 -19529.642} C_VEL
LIN {X 0,Y 319.965,Z 1071.429,A -85,B 0,C 180,E1 -19533.583,E2 -19533.583} C_VEL
LIN {X 0,Y 319.992,Z 1069.709,A -85,B 0,C 180,E1 -19537.18,E2 -19537.18} C_VEL
LIN {X 0,Y 320.245,Z 1066.887,A -85,B 0,C 180,E1 -19540.797,E2 -19540.797} C_VEL
LIN {X 0,Y 321.202,Z 1062.031,A -85,B 0,C 180,E1 -19545.158,E2 -19545.158} C_VEL
LIN {X 0,Y 323.026,Z 1055.636,A -85,B 0,C 180,E1 -19549.342,E2 -19549.342} C_VEL
LIN {X 0,Y 325.959,Z 1047.736,A -85,B 0,C 180,E1 -19553.502,E2 -19553.502} C_VEL
LIN {X 0,Y 330.124,Z 1037.883,A -85,B 0,C 180,E1 -19557.607,E2 -19557.607} C_VEL
LIN {X 0,Y 335.362,Z 1026.831,A -85,B 0,C 180,E1 -19561.451,E2 -19561.451} C_VEL
LIN {X 0,Y 341.509,Z 1014.301,A -85,B 0,C 180,E1 -19565.02,E2 -19565.02} C_VEL
LIN {X 0,Y 348.055,Z 1001.369,A -85,B 0,C 180,E1 -19568.145,E2 -19568.145} C_VEL
LIN {X 0,Y 355.914,Z 985.696,A -85,B 0,C 180,E1 -19571.315,E2 -19571.315} C_VEL
LIN {X 0,Y 363.373,Z 970.519,A -85,B 0,C 180,E1 -19573.902,E2 -19573.902} C_VEL
LIN {X 0,Y 372.53,Z 951.131,A -85,B 0,C 180,E1 -19576.667,E2 -19576.667} C_VEL
LIN {X 0,Y 379.927,Z 934.488,A -85,B 0,C 180,E1 -19578.656,E2 -19578.656} C_VEL
LIN {X 0,Y 388.334,Z 914.306,A -85,B 0,C 180,E1 -19580.698,E2 -19580.698} C_VEL
LIN {X 0,Y 395.546,Z 895.237,A -85,B 0,C 180,E1 -19582.3,E2 -19582.3} C_VEL
LIN {X 0,Y 402.808,Z 874.339,A -85,B 0,C 180,E1 -19583.779,E2 -19583.779} C_VEL
LIN {X 0,Y 409.482,Z 852.2,A -85,B 0,C 180,E1 -19585.058,E2 -19585.058} C_VEL
LIN {X 0,Y 414.821,Z 832.068,A -85,B 0,C 180,E1 -19586.015,E2 -19586.015} C_VEL
LIN {X 0,Y 420.549,Z 806.33,A -85,B 0,C 180,E1 -19586.979,E2 -19586.979} C_VEL
LIN {X 0,Y 424.429,Z 784.485,A -85,B 0,C 180,E1 -19587.602,E2 -19587.602} C_VEL
LIN {X 0,Y 427.844,Z 757.345,A -85,B 0,C 180,E1 -19588.186,E2 -19588.186} C_VEL
LIN {X 0,Y 444.04,Z 530.249,A -85,B 0,C 180,E1 -19591.884,E2 -19591.884} C_VEL
LIN {X 0,Y 444.054,Z 528.336,A -85,B 0,C 180,E1 -19591.944,E2 -19591.944} C_VEL
LIN {X 0,Y 436.387,Z 513.786,A -85,B 0,C 180,E1 -19594.411,E2 -19594.411} C_VEL
LIN {X 0,Y 428.718,Z 500.151,A -85,B 0,C 180,E1 -19597.186,E2 -19597.186} C_VEL
LIN {X 0,Y 421.533,Z 488.355,A -85,B 0,C 180,E1 -19600.172,E2 -19600.172} C_VEL
LIN {X 0,Y 417.444,Z 482.738,A -85,B 0,C 180,E1 -19602.074,E2 -19602.074} C_VEL
LIN {X 0,Y 414.367,Z 478.485,A -85,B 0,C 180,E1 -19603.673,E2 -19603.673} C_VEL
LIN {X 0,Y 411.026,Z 473.855,A -85,B 0,C 180,E1 -19605.633,E2 -19605.633} C_VEL
LIN {X 0,Y 407.46,Z 468.936,A -85,B 0,C 180,E1 -19608.104,E2 -19608.104} C_VEL
LIN {X 0,Y 404.231,Z 464.888,A -85,B 0,C 180,E1 -19610.891,E2 -19610.891} C_VEL
LIN {X 0,Y 403.347,Z 463.326,A -85,B 0,C 180,E1 -19611.877,E2 -19611.877} C_VEL
LIN {X 0,Y 399.874,Z 458.51,A -85,B 0,C 180,E1 -19618.424,E2 -19618.424} C_VEL
LIN {X 0,Y 399.815,Z 457.428,A -85,B 0,C 180,E1 -19620.43,E2 -19620.43} C_VEL
LIN {X 0,Y 403.354,Z 463.351,A -85,B 0,C 180,E1 -19628.554,E2 -19628.554} C_VEL
LIN {X 0,Y 403.984,Z 464.385,A -85,B 0,C 180,E1 -19629.258,E2 -19629.258} C_VEL
LIN {X 0,Y 406.733,Z 468.295,A -85,B 0,C 180,E1 -19631.774,E2 -19631.774} C_VEL
LIN {X 0,Y 407.932,Z 469.571,A -85,B 0,C 180,E1 -19632.672,E2 -19632.672} C_VEL
LIN {X 0,Y 411.269,Z 474.116,A -85,B 0,C 180,E1 -19634.934,E2 -19634.934} C_VEL
LIN {X 0,Y 416.029,Z 480.702,A -85,B 0,C 180,E1 -19637.628,E2 -19637.628} C_VEL
LIN {X 0,Y 420.312,Z 486.755,A -85,B 0,C 180,E1 -19639.707,E2 -19639.707} C_VEL
LIN {X 0,Y 425.852,Z 494.631,A -85,B 0,C 180,E1 -19642.066,E2 -19642.066} C_VEL
LIN {X 0,Y 433.365,Z 505.944,A -85,B 0,C 180,E1 -19644.866,E2 -19644.866} C_VEL
LIN {X 0,Y 441.748,Z 519.484,A -85,B 0,C 180,E1 -19647.61,E2 -19647.61} C_VEL
LIN {X 0,Y 444.326,Z 524.047,A -85,B 0,C 180,E1 -19648.398,E2 -19648.398} C_VEL
LIN {X 0,Y 428.431,Z 745.763,A -85,B 0,C 180,E1 -19652.003,E2 -19652.003} C_VEL
LIN {X 0,Y 425.136,Z 772.429,A -85,B 0,C 180,E1 -19652.6,E2 -19652.6} C_VEL
LIN {X 0,Y 421.643,Z 793.01,A -85,B 0,C 180,E1 -19653.22,E2 -19653.22} C_VEL
LIN {X 0,Y 416.694,Z 816.604,A -85,B 0,C 180,E1 -19654.121,E2 -19654.121} C_VEL
LIN {X 0,Y 411.383,Z 837.325,A -85,B 0,C 180,E1 -19655.118,E2 -19655.118} C_VEL
LIN {X 0,Y 405.266,Z 858.318,A -85,B 0,C 180,E1 -19656.336,E2 -19656.336} C_VEL
LIN {X 0,Y 397.834,Z 880.329,A -85,B 0,C 180,E1 -19657.891,E2 -19657.891} C_VEL
LIN {X 0,Y 391.003,Z 898.674,A -85,B 0,C 180,E1 -19659.44,E2 -19659.44} C_VEL
LIN {X 0,Y 382.292,Z 919.882,A -85,B 0,C 180,E1 -19661.58,E2 -19661.58} C_VEL
LIN {X 0,Y 374.769,Z 936.769,A -85,B 0,C 180,E1 -19663.612,E2 -19663.612} C_VEL
LIN {X 0,Y 365.973,Z 955.357,A -85,B 0,C 180,E1 -19666.273,E2 -19666.273} C_VEL
LIN {X 0,Y 358.481,Z 970.337,A -85,B 0,C 180,E1 -19668.833,E2 -19668.833} C_VEL
LIN {X 0,Y 350.528,Z 985.844,A -85,B 0,C 180,E1 -19671.965,E2 -19671.965} C_VEL
LIN {X 0,Y 343.685,Z 998.84,A -85,B 0,C 180,E1 -19675.128,E2 -19675.128} C_VEL
LIN {X 0,Y 337.23,Z 1011.386,A -85,B 0,C 180,E1 -19678.743,E2 -19678.743} C_VEL
LIN {X 0,Y 331.776,Z 1022.113,A -85,B 0,C 180,E1 -19682.542,E2 -19682.542} C_VEL
LIN {X 0,Y 327.343,Z 1031.653,A -85,B 0,C 180,E1 -19686.604,E2 -19686.604} C_VEL
LIN {X 0,Y 324.093,Z 1039.3,A -85,B 0,C 180,E1 -19690.748,E2 -19690.748} C_VEL
LIN {X 0,Y 322.043,Z 1045.15,A -85,B 0,C 180,E1 -19694.698,E2 -19694.698} C_VEL
LIN {X 0,Y 320.712,Z 1049.976,A -85,B 0,C 180,E1 -19699.139,E2 -19699.139} C_VEL
LIN {X 0,Y 320.21,Z 1052.728,A -85,B 0,C 180,E1 -19702.825,E2 -19702.825} C_VEL
LIN {X 0,Y 320.017,Z 1054.497,A -85,B 0,C 180,E1 -19706.776,E2 -19706.776} C_VEL
LIN {X 0,Y 319.992,Z 1054.869,A -85,B 0,C 180,E1 -19710.895,E2 -19710.895} C_VEL
LIN {X 0,Y 320.054,Z 1054.074,A -85,B 0,C 180,E1 -19714.48,E2 -19714.48} C_VEL
LIN {X 0,Y 320.279,Z 1052.246,A -85,B 0,C 180,E1 -19718.076,E2 -19718.076} C_VEL
LIN {X 0,Y 321.102,Z 1048.428,A -85,B 0,C 180,E1 -19722.59,E2 -19722.59} C_VEL
LIN {X 0,Y 322.473,Z 1043.811,A -85,B 0,C 180,E1 -19726.39,E2 -19726.39} C_VEL
LIN {X 0,Y 324.918,Z 1037.369,A -85,B 0,C 180,E1 -19730.538,E2 -19730.538} C_VEL
LIN {X 0,Y 328.478,Z 1029.12,A -85,B 0,C 180,E1 -19734.647,E2 -19734.647} C_VEL
LIN {X 0,Y 332.809,Z 1020.125,A -85,B 0,C 180,E1 -19738.34,E2 -19738.34} C_VEL
LIN {X 0,Y 338.792,Z 1008.354,A -85,B 0,C 180,E1 -19742.289,E2 -19742.289} C_VEL
LIN {X 0,Y 344.701,Z 997.029,A -85,B 0,C 180,E1 -19745.461,E2 -19745.461} C_VEL
LIN {X 0,Y 352.75,Z 981.666,A -85,B 0,C 180,E1 -19749.043,E2 -19749.043} C_VEL
LIN {X 0,Y 360.018,Z 967.478,A -85,B 0,C 180,E1 -19751.802,E2 -19751.802} C_VEL
LIN {X 0,Y 369.051,Z 949.149,A -85,B 0,C 180,E1 -19754.784,E2 -19754.784} C_VEL
LIN {X 0,Y 376.525,Z 933.154,A -85,B 0,C 180,E1 -19756.962,E2 -19756.962} C_VEL
LIN {X 0,Y 385.32,Z 913.067,A -85,B 0,C 180,E1 -19759.264,E2 -19759.264} C_VEL
LIN {X 0,Y 392.679,Z 894.657,A -85,B 0,C 180,E1 -19761.027,E2 -19761.027} C_VEL
LIN {X 0,Y 400.286,Z 873.868,A -85,B 0,C 180,E1 -19762.711,E2 -19762.711} C_VEL
LIN {X 0,Y 406.878,Z 853.424,A -85,B 0,C 180,E1 -19764.07,E2 -19764.07} C_VEL
LIN {X 0,Y 408.694,Z 847.523,A -85,B 0,C 180,E1 -19764.425,E2 -19764.425} C_VEL
LIN {X 0,Y 410.121,Z 840.778,A -85,B 0,C 180,E1 -19764.925,E2 -19764.925} C_VEL
LIN {X 0,Y 411.25,Z 823.017,A -85,B 0,C 180,E1 -19766.537,E2 -19766.537} C_VEL
LIN {X 0,Y 412.356,Z 817.004,A -85,B 0,C 180,E1 -19766.9,E2 -19766.9} C_VEL
LIN {X 0,Y 417.486,Z 793.136,A -85,B 0,C 180,E1 -19767.808,E2 -19767.808} C_VEL
LIN {X 0,Y 421.05,Z 772.594,A -85,B 0,C 180,E1 -19768.424,E2 -19768.424} C_VEL
LIN {X 0,Y 424.417,Z 745.929,A -85,B 0,C 180,E1 -19769.018,E2 -19769.018} C_VEL
LIN {X 0,Y 440.451,Z 528.429,A -85,B 0,C 180,E1 -19772.553,E2 -19772.553} C_VEL
LIN {X 0,Y 433.278,Z 516.5,A -85,B 0,C 180,E1 -19774.91,E2 -19774.91} C_VEL
LIN {X 0,Y 426.217,Z 505.341,A -85,B 0,C 180,E1 -19777.518,E2 -19777.518} C_VEL
LIN {X 0,Y 419.645,Z 495.656,A -85,B 0,C 180,E1 -19780.296,E2 -19780.296} C_VEL
LIN {X 0,Y 415.679,Z 490.029,A -85,B 0,C 180,E1 -19782.212,E2 -19782.212} C_VEL
LIN {X 0,Y 412.944,Z 486.106,A -85,B 0,C 180,E1 -19783.687,E2 -19783.687} C_VEL
LIN {X 0,Y 409.794,Z 481.713,A -85,B 0,C 180,E1 -19785.589,E2 -19785.589} C_VEL
LIN {X 0,Y 406.148,Z 476.637,A -85,B 0,C 180,E1 -19788.209,E2 -19788.209} C_VEL
LIN {X 0,Y 403.27,Z 472.988,A -85,B 0,C 180,E1 -19790.797,E2 -19790.797} C_VEL
LIN {X 0,Y 402.366,Z 471.289,A -85,B 0,C 180,E1 -19791.857,E2 -19791.857} C_VEL
LIN {X 0,Y 399.066,Z 466.49,A -85,B 0,C 180,E1 -19799.569,E2 -19799.569} C_VEL
LIN {X 0,Y 399.206,Z 467.355,A -85,B 0,C 180,E1 -19801.866,E2 -19801.866} C_VEL
LIN {X 0,Y 402.651,Z 471.63,A -85,B 0,C 180,E1 -19808.137,E2 -19808.137} C_VEL
LIN {X 0,Y 405.492,Z 476.021,A -85,B 0,C 180,E1 -19810.945,E2 -19810.945} C_VEL
LIN {X 0,Y 406.847,Z 477.594,A -85,B 0,C 180,E1 -19812.009,E2 -19812.009} C_VEL
LIN {X 0,Y 410.721,Z 482.98,A -85,B 0,C 180,E1 -19814.666,E2 -19814.666} C_VEL
LIN {X 0,Y 414.857,Z 488.841,A -85,B 0,C 180,E1 -19817.028,E2 -19817.028} C_VEL
LIN {X 0,Y 418.733,Z 494.339,A -85,B 0,C 180,E1 -19818.951,E2 -19818.951} C_VEL
LIN {X 0,Y 421.814,Z 499.214,A -85,B 0,C 180,E1 -19820.357,E2 -19820.357} C_VEL
LIN {X 0,Y 428.443,Z 510.551,A -85,B 0,C 180,E1 -19823.084,E2 -19823.084} C_VEL
LIN {X 0,Y 436.136,Z 524.727,A -85,B 0,C 180,E1 -19825.86,E2 -19825.86} C_VEL
LIN {X 0,Y 440.262,Z 533.057,A -85,B 0,C 180,E1 -19827.23,E2 -19827.23} C_VEL
LIN {X 0,Y 423.798,Z 757.465,A -85,B 0,C 180,E1 -19830.883,E2 -19830.883} C_VEL
LIN {X 0,Y 420.318,Z 784.397,A -85,B 0,C 180,E1 -19831.462,E2 -19831.462} C_VEL
LIN {X 0,Y 416.355,Z 806.216,A -85,B 0,C 180,E1 -19832.082,E2 -19832.082} C_VEL
LIN {X 0,Y 410.732,Z 831.038,A -85,B 0,C 180,E1 -19833.001,E2 -19833.001} C_VEL
LIN {X 0,Y 405.125,Z 851.717,A -85,B 0,C 180,E1 -19833.975,E2 -19833.975} C_VEL
LIN {X 0,Y 398.411,Z 873.537,A -85,B 0,C 180,E1 -19835.224,E2 -19835.224} C_VEL
LIN {X 0,Y 390.953,Z 894.495,A -85,B 0,C 180,E1 -19836.698,E2 -19836.698} C_VEL
LIN {X 0,Y 383.504,Z 913.663,A -85,B 0,C 180,E1 -19838.299,E2 -19838.299} C_VEL
LIN {X 0,Y 374.717,Z 934.189,A -85,B 0,C 180,E1 -19840.375,E2 -19840.375} C_VEL
LIN {X 0,Y 367.216,Z 950.536,A -85,B 0,C 180,E1 -19842.331,E2 -19842.331} C_VEL
LIN {X 0,Y 357.976,Z 969.513,A -85,B 0,C 180,E1 -19845.035,E2 -19845.035} C_VEL
LIN {X 0,Y 350.198,Z 984.754,A -85,B 0,C 180,E1 -19847.636,E2 -19847.636} C_VEL
LIN {X 0,Y 341.968,Z 1000.545,A -85,B 0,C 180,E1 -19850.834,E2 -19850.834} C_VEL
LIN {X 0,Y 335.095,Z 1013.526,A -85,B 0,C 180,E1 -19853.997,E2 -19853.997} C_VEL
LIN {X 0,Y 328.602,Z 1026.142,A -85,B 0,C 180,E1 -19857.619,E2 -19857.619} C_VEL
LIN {X 0,Y 323.038,Z 1037.255,A -85,B 0,C 180,E1 -19861.532,E2 -19861.532} C_VEL
LIN {X 0,Y 318.729,Z 1046.765,A -85,B 0,C 180,E1 -19865.537,E2 -19865.537} C_VEL
LIN {X 0,Y 315.499,Z 1054.837,A -85,B 0,C 180,E1 -19869.791,E2 -19869.791} C_VEL
LIN {X 0,Y 313.581,Z 1060.804,A -85,B 0,C 180,E1 -19873.704,E2 -19873.704} C_VEL
LIN {X 0,Y 312.363,Z 1066.217,A -85,B 0,C 180,E1 -19878.386,E2 -19878.386} C_VEL
LIN {X 0,Y 311.998,Z 1069.274,A -85,B 0,C 180,E1 -19882.264,E2 -19882.264} C_VEL
LIN {X 0,Y 311.962,Z 1071.014,A -85,B 0,C 180,E1 -19885.772,E2 -19885.772} C_VEL
LIN {X 0,Y 311.988,Z 1071.775,A -85,B 0,C 180,E1 -19889.449,E2 -19889.449} C_VEL
LIN {X 0,Y 311.968,Z 1071.285,A -85,B 0,C 180,E1 -19893.491,E2 -19893.491} C_VEL
LIN {X 0,Y 311.998,Z 1069.494,A -85,B 0,C 180,E1 -19897.365,E2 -19897.365} C_VEL
LIN {X 0,Y 312.281,Z 1066.671,A -85,B 0,C 180,E1 -19901.076,E2 -19901.076} C_VEL
LIN {X 0,Y 313.317,Z 1061.812,A -85,B 0,C 180,E1 -19905.549,E2 -19905.549} C_VEL
LIN {X 0,Y 315.277,Z 1055.415,A -85,B 0,C 180,E1 -19909.837,E2 -19909.837} C_VEL
LIN {X 0,Y 318.401,Z 1047.515,A -85,B 0,C 180,E1 -19914.094,E2 -19914.094} C_VEL
LIN {X 0,Y 322.807,Z 1037.66,A -85,B 0,C 180,E1 -19918.289,E2 -19918.289} C_VEL
LIN {X 0,Y 328.311,Z 1026.608,A -85,B 0,C 180,E1 -19922.206,E2 -19922.206} C_VEL
LIN {X 0,Y 334.749,Z 1014.078,A -85,B 0,C 180,E1 -19925.835,E2 -19925.835} C_VEL
LIN {X 0,Y 341.57,Z 1001.146,A -85,B 0,C 180,E1 -19929.004,E2 -19929.004} C_VEL
LIN {X 0,Y 349.856,Z 985.255,A -85,B 0,C 180,E1 -19932.249,E2 -19932.249} C_VEL
LIN {X 0,Y 357.476,Z 970.296,A -85,B 0,C 180,E1 -19934.818,E2 -19934.818} C_VEL
LIN {X 0,Y 366.935,Z 950.908,A -85,B 0,C 180,E1 -19937.601,E2 -19937.601} C_VEL
LIN {X 0,Y 374.417,Z 934.588,A -85,B 0,C 180,E1 -19939.561,E2 -19939.561} C_VEL
LIN {X 0,Y 382.908,Z 914.857,A -85,B 0,C 180,E1 -19941.575,E2 -19941.575} C_VEL
LIN {X 0,Y 390.62,Z 895.014,A -85,B 0,C 180,E1 -19943.245,E2 -19943.245} C_VEL
LIN {X 0,Y 398.065,Z 874.117,A -85,B 0,C 180,E1 -19944.722,E2 -19944.722} C_VEL
LIN {X 0,Y 404.907,Z 851.963,A -85,B 0,C 180,E1 -19945.997,E2 -19945.997} C_VEL
LIN {X 0,Y 410.366,Z 831.845,A -85,B 0,C 180,E1 -19946.949,E2 -19946.949} C_VEL
LIN {X 0,Y 416.198,Z 806.213,A -85,B 0,C 180,E1 -19947.904,E2 -19947.904} C_VEL
LIN {X 0,Y 420.157,Z 784.388,A -85,B 0,C 180,E1 -19948.524,E2 -19948.524} C_VEL
LIN {X 0,Y 423.655,Z 757.218,A -85,B 0,C 180,E1 -19949.108,E2 -19949.108} C_VEL
LIN {X 0,Y 440.095,Z 532.853,A -85,B 0,C 180,E1 -19952.761,E2 -19952.761} C_VEL
LIN {X 0,Y 433.807,Z 520.512,A -85,B 0,C 180,E1 -19954.869,E2 -19954.869} C_VEL
LIN {X 0,Y 426.388,Z 507.028,A -85,B 0,C 180,E1 -19957.636,E2 -19957.636} C_VEL
LIN {X 0,Y 419.516,Z 495.525,A -85,B 0,C 180,E1 -19960.58,E2 -19960.58} C_VEL
LIN {X 0,Y 415.526,Z 489.925,A -85,B 0,C 180,E1 -19962.495,E2 -19962.495} C_VEL
LIN {X 0,Y 412.772,Z 486.03,A -85,B 0,C 180,E1 -19963.969,E2 -19963.969} C_VEL
LIN {X 0,Y 409.502,Z 481.429,A -85,B 0,C 180,E1 -19965.939,E2 -19965.939} C_VEL
LIN {X 0,Y 406.117,Z 476.662,A -85,B 0,C 180,E1 -19968.352,E2 -19968.352} C_VEL
LIN {X 0,Y 402.916,Z 472.448,A -85,B 0,C 180,E1 -19971.221,E2 -19971.221} C_VEL
LIN {X 0,Y 402.244,Z 471.211,A -85,B 0,C 180,E1 -19971.998,E2 -19971.998} C_VEL
LIN {X 0,Y 398.877,Z 466.387,A -85,B 0,C 180,E1 -19978.564,E2 -19978.564} C_VEL
